	#internal.panel[#PB_Configuration.itLoaderPbID].boSemiAMode := #internal.boManSelOnPressL OR #internal.boSetupSelOnPressL OR #internal.boManSelOnPressR OR #internal.boSetupSelOnPressR;
	#internal.panel[#PB_Configuration.itGTSPbID].boSemiAMode := #internal.boManSelOnPressL OR #internal.boSetupSelOnPressL OR #internal.boManSelOnPressR OR #internal.boSetupSelOnPressR;
	#internal.panel[#PB_Configuration.itPressPbID].boSemiAMode := #internal.boManSelOnPressL OR #internal.boSetupSelOnPressL OR #internal.boManSelOnPressR OR #internal.boSetupSelOnPressR;
	#internal.panel[#PB_Configuration.itSegmentsPbID].boSemiAMode := #internal.boManSelOnPressL OR #internal.boSetupSelOnPressL OR #internal.boManSelOnPressR OR #internal.boSetupSelOnPressR;
	#internal.panel[#PB_Configuration.itSqueezePbID].boSemiAMode := #internal.boManSelOnPressL OR #internal.boSetupSelOnPressL OR #internal.boManSelOnPressR OR #internal.boSetupSelOnPressR;
	#internal.panel[#PB_Configuration.itTopRingPbID].boSemiAMode := #internal.boManSelOnPressL OR #internal.boSetupSelOnPressL OR #internal.boManSelOnPressR OR #internal.boSetupSelOnPressR;
	#internal.panel[#PB_Configuration.itBotRingPbID].boSemiAMode := #internal.boManSelOnPressL OR #internal.boSetupSelOnPressL OR #internal.boManSelOnPressR OR #internal.boSetupSelOnPressR;
	#internal.panel[#PB_Configuration.itBeadRingPbID].boSemiAMode := #internal.boManSelOnPressL OR #internal.boSetupSelOnPressL OR #internal.boManSelOnPressR OR #internal.boSetupSelOnPressR;
	#internal.panel[#PB_Configuration.itUnloaderPbID].boSemiAMode := #internal.boManSelOnPressL OR #internal.boSetupSelOnPressL OR #internal.boManSelOnPressR OR #internal.boSetupSelOnPressR;
	#internal.panel[#PB_Configuration.itUnloaderPCIPbID].boSemiAMode := #internal.boManSelOnPressL OR #internal.boSetupSelOnPressL OR #internal.boManSelOnPressR OR #internal.boSetupSelOnPressR;
	#internal.panel[#PB_Configuration.itExitConvPbId].boSemiAMode := #internal.boManSelOnPressL OR #internal.boSetupSelOnPressL OR #internal.boManSelOnPressR OR #internal.boSetupSelOnPressR;
	#internal.panel[#PB_Configuration.itHPUPbID].boSemiAMode := (#internal.boManSelOnPressL OR #internal.boSetupSelOnPressL) AND (#internal.boManSelOnPressR OR #internal.boSetupSelOnPressR);
	#internal.panel[#PB_Configuration.itLoaderPbID].boAutoMode := NOT #internal.panel[#PB_Configuration.itLoaderPbID].boSemiAMode;
	#internal.panel[#PB_Configuration.itGTSPbID].boAutoMode := NOT #internal.panel[#PB_Configuration.itGTSPbID].boSemiAMode;
	#internal.panel[#PB_Configuration.itPressPbID].boAutoMode := NOT #internal.panel[#PB_Configuration.itPressPbID].boSemiAMode;
	#internal.panel[#PB_Configuration.itSegmentsPbID].boAutoMode := NOT #internal.panel[#PB_Configuration.itSegmentsPbID].boSemiAMode;
	#internal.panel[#PB_Configuration.itSqueezePbID].boAutoMode := NOT #internal.panel[#PB_Configuration.itSqueezePbID].boSemiAMode;
	#internal.panel[#PB_Configuration.itTopRingPbID].boAutoMode := NOT #internal.panel[#PB_Configuration.itTopRingPbID].boSemiAMode;
	#internal.panel[#PB_Configuration.itBotRingPbID].boAutoMode := NOT #internal.panel[#PB_Configuration.itBotRingPbID].boSemiAMode;
	#internal.panel[#PB_Configuration.itBeadRingPbID].boAutoMode := NOT #internal.panel[#PB_Configuration.itBeadRingPbID].boSemiAMode;
	#internal.panel[#PB_Configuration.itUnloaderPbID].boAutoMode := NOT #internal.panel[#PB_Configuration.itUnloaderPbID].boSemiAMode;
	#internal.panel[#PB_Configuration.itUnloaderPCIPbID].boAutoMode := NOT #internal.panel[#PB_Configuration.itUnloaderPCIPbID].boSemiAMode;
	#internal.panel[#PB_Configuration.itExitConvPbId].boAutoMode := NOT #internal.panel[#PB_Configuration.itExitConvPbId].boSemiAMode;
	#internal.panel[#PB_Configuration.itHPUPbID].boAutoMode := NOT #internal.panel[#PB_Configuration.itHPUPbID].boSemiAMode;
	#internal.panel[#PB_Configuration.itShapingPbID].boSemiAMode := #internal.boManSelOnHeatingL OR #internal.boSetupSelOnHeatingL OR #internal.boManSelOnHeatingR OR #internal.boSetupSelOnHeatingR;
	#internal.panel[#PB_Configuration.itDrainPbID].boSemiAMode := #internal.boManSelOnHeatingL OR #internal.boSetupSelOnHeatingL OR #internal.boManSelOnHeatingR OR #internal.boSetupSelOnHeatingR;
	#internal.panel[#PB_Configuration.itVacuumPbID].boSemiAMode := #internal.boManSelOnHeatingL OR #internal.boSetupSelOnHeatingL OR #internal.boManSelOnHeatingR OR #internal.boSetupSelOnHeatingR;
	#internal.panel[#PB_Configuration.itExtHeatingPbID].boSemiAMode := #internal.boManSelOnHeatingL OR #internal.boSetupSelOnHeatingL OR #internal.boManSelOnHeatingR OR #internal.boSetupSelOnHeatingR;
	#internal.panel[#PB_Configuration.itShapingPbID].boAutoMode := NOT #internal.panel[#PB_Configuration.itShapingPbID].boSemiAMode;
	#internal.panel[#PB_Configuration.itDrainPbID].boAutoMode := NOT #internal.panel[#PB_Configuration.itDrainPbID].boSemiAMode;
	#internal.panel[#PB_Configuration.itVacuumPbID].boAutoMode := NOT #internal.panel[#PB_Configuration.itVacuumPbID].boSemiAMode;
	#internal.panel[#PB_Configuration.itExtHeatingPbID].boAutoMode := NOT #internal.panel[#PB_Configuration.itExtHeatingPbID].boSemiAMode;
	END_REGION

	//=======================================================================================================================================
	//            READ INPUTS FROM KP32F
	//=======================================================================================================================================
	REGION READ INPUTS FROM KP32F
	    // Enable test lamp button
	    #internal.panel[#PB_Configuration.itLampTestPbID].boEnable := TRUE;

	    IF NOT "SYS_SimulationActive" THEN
	        // Read push buttons from 0 to 15
	        #readWriteData(itDeviceNumber := #itKP32DeviceNumber,
	                       uiPNIO_SysID := #uiPNIOSysID,
	                       uiSlotNumber := 1,
	                       uiSubSlotNumber := 0,
	                       bo0read_1write := FALSE,
	                       vaModuleSlotData := #internal.buttons0_15);
	        // Read push buttons from 16 to 31
	        #readWriteData(itDeviceNumber := #itKP32DeviceNumber,
	                       uiPNIO_SysID := #uiPNIOSysID,
	                       uiSlotNumber := 2,
	                       uiSubSlotNumber := 0,
	                       bo0read_1write := FALSE,
	                       vaModuleSlotData := #internal.buttons16_31);
	    END_IF;

	    // KP32F management of lamps and buttons
	    FOR #itPushButtonIndexTemp := 0 TO 31 DO

	        (*
	        Push buttons lamp management:
	                OUT:   red      green      blue
	        COLOUR:
	            red         1         0         0
	            green       0         1         0
	            blue        0         0         1
	            yellow      1         1         0
	            white       1         1         1
	            OFF         0         0         0
	            OFF         0         1         1
	            OFF         1         0         1

	        Push buttons order in the panel:
	            07  06  05  04  03  02  01  00
	            15  14  13  12  11  10  09  08
	            23  22  21  20  19  18  17  16
	            31  30  29  28  27  26  25  24
	        *)
	        // Read command button
	        IF NOT "SYS_SimulationActive" THEN
	            CASE #itPushButtonIndexTemp OF
	                0:
	                    #internal.panel[#itPushButtonIndexTemp].boCmdOn := #internal.buttons0_15.PB00;
	                1:
	                    #internal.panel[#itPushButtonIndexTemp].boCmdOn := #internal.buttons0_15.PB01;
	                2:
	                    #internal.panel[#itPushButtonIndexTemp].boCmdOn := #internal.buttons0_15.PB02;
	                3:
	                    #internal.panel[#itPushButtonIndexTemp].boCmdOn := #internal.buttons0_15.PB03;
	                4:
	                    #internal.panel[#itPushButtonIndexTemp].boCmdOn := #internal.buttons0_15.PB04;
	                5:
	                    #internal.panel[#itPushButtonIndexTemp].boCmdOn := #internal.buttons0_15.PB05;
	                6:
	                    #internal.panel[#itPushButtonIndexTemp].boCmdOn := #internal.buttons0_15.PB06;
	                7:
	                    #internal.panel[#itPushButtonIndexTemp].boCmdOn := #internal.buttons0_15.PB07;
	                8:
	                    #internal.panel[#itPushButtonIndexTemp].boCmdOn := #internal.buttons0_15.PB08;
	                9:
	                    #internal.panel[#itPushButtonIndexTemp].boCmdOn := #internal.buttons0_15.PB09;
	                10:
	                    #internal.panel[#itPushButtonIndexTemp].boCmdOn := #internal.buttons0_15.PB10;
	                11:
	                    #internal.panel[#itPushButtonIndexTemp].boCmdOn := #internal.buttons0_15.PB11;
	                12:
	                    #internal.panel[#itPushButtonIndexTemp].boCmdOn := #internal.buttons0_15.PB12;
	                13:
	                    #internal.panel[#itPushButtonIndexTemp].boCmdOn := #internal.buttons0_15.PB13;
	                14:
	                    #internal.panel[#itPushButtonIndexTemp].boCmdOn := #internal.buttons0_15.PB14;
	                15:
	                    #internal.panel[#itPushButtonIndexTemp].boCmdOn := #internal.buttons0_15.PB15;
	                16:
	                    #internal.panel[#itPushButtonIndexTemp].boCmdOn := #internal.buttons16_31.PB16;
	                17:
	                    #internal.panel[#itPushButtonIndexTemp].boCmdOn := #internal.buttons16_31.PB17;
	                18:
	                    #internal.panel[#itPushButtonIndexTemp].boCmdOn := #internal.buttons16_31.PB18;
	                19:
	                    #internal.panel[#itPushButtonIndexTemp].boCmdOn := #internal.buttons16_31.PB19;
	                20:
	                    #internal.panel[#itPushButtonIndexTemp].boCmdOn := #internal.buttons16_31.PB20;
	                21:
	                    #internal.panel[#itPushButtonIndexTemp].boCmdOn := #internal.buttons16_31.PB21;
	                22:
	                    #internal.panel[#itPushButtonIndexTemp].boCmdOn := #internal.buttons16_31.PB22;
	                23:
	                    #internal.panel[#itPushButtonIndexTemp].boCmdOn := #internal.buttons16_31.PB23;
	                24:
	                    #internal.panel[#itPushButtonIndexTemp].boCmdOn := #internal.buttons16_31.PB24;
	                25:
	                    #internal.panel[#itPushButtonIndexTemp].boCmdOn := #internal.buttons16_31.PB25;
	                26:
	                    #internal.panel[#itPushButtonIndexTemp].boCmdOn := #internal.buttons16_31.PB26;
	                27:
	                    #internal.panel[#itPushButtonIndexTemp].boCmdOn := #internal.buttons16_31.PB27;
	                28:
	                    #internal.panel[#itPushButtonIndexTemp].boCmdOn := #internal.buttons16_31.PB28;
	                29:
	                    #internal.panel[#itPushButtonIndexTemp].boCmdOn := #internal.buttons16_31.PB29;
	                30:
	                    #internal.panel[#itPushButtonIndexTemp].boCmdOn := #internal.buttons16_31.PB30;
	                31:
	                    #internal.panel[#itPushButtonIndexTemp].boCmdOn := #internal.buttons16_31.PB31;
	                ELSE
	                    #internal.panel[#itPushButtonIndexTemp].boCmdOn := FALSE;
	            END_CASE;
	        ELSE
	            #internal.panel[#itPushButtonIndexTemp].boCmdOn := #internal.simulation[#itPushButtonIndexTemp].boPB;
	        END_IF;
	        #internal.panel[#itPushButtonIndexTemp].boCmdWrong := FALSE;
	        IF NOT #internal.panel[#itPushButtonIndexTemp].boEnable OR #boChgOfModeFiltTemp THEN
	            IF #internal.panel[#itPushButtonIndexTemp].boCmdOn AND NOT #boChgOfModeFiltTemp THEN
	                #internal.panel[#itPushButtonIndexTemp].boCmdWrong := TRUE;
	                #boWrongPushCmdTemp := TRUE;
	            END_IF;
	            #internal.panel[#itPushButtonIndexTemp].boCmdOn := FALSE;
	            #internal.panel[#itPushButtonIndexTemp].boSelect := FALSE;
	        END_IF;
	        #internal.panel[#itPushButtonIndexTemp].boCmdRE := #internal.panel[#itPushButtonIndexTemp].boCmdOn AND NOT #internal.panel[#itPushButtonIndexTemp].boCmdMem;
	        #internal.panel[#itPushButtonIndexTemp].boCmdFE := NOT #internal.panel[#itPushButtonIndexTemp].boCmdOn AND #internal.panel[#itPushButtonIndexTemp].boCmdMem;
	        #internal.panel[#itPushButtonIndexTemp].boCmdMem := #internal.panel[#itPushButtonIndexTemp].boCmdOn;

	        IF (#internal.panel[#itPushButtonIndexTemp].itPBType = #PB_EQUIPMENT) AND #internal.panel[#itPushButtonIndexTemp].boCmdRE THEN
	            #internal.panel[#itPushButtonIndexTemp].boSelect := NOT #internal.panel[#itPushButtonIndexTemp].boSelect;
	            FOR #itPushButtonIndex2Temp := 0 TO 31 DO
	                IF (#internal.panel[#itPushButtonIndex2Temp].itPBType = #PB_EQUIPMENT) AND (#itPushButtonIndexTemp <> #itPushButtonIndex2Temp) THEN
	                    #internal.panel[#itPushButtonIndex2Temp].boSelect := FALSE;
	                END_IF;
	            END_FOR;
	            #boResetPBsStatesTemp := TRUE;
	        END_IF;

	    END_FOR;
	END_REGION


	//=======================================================================================================================================
	//            CAVITY SELECTION
	//=======================================================================================================================================
	REGION CAVITY SELECTION
	    #internal.panel[#PB_Configuration.itLeftSelPbID].boEnable := TRUE;
	    #internal.panel[#PB_Configuration.itRightSelPbID].boEnable := TRUE;
	    #internal.panel[#PB_Configuration.itLeftSelPbID].boAborted := FALSE;
	    #internal.panel[#PB_Configuration.itRightSelPbID].boAborted := FALSE;
	    #internal.panel[#PB_Configuration.itLeftSelPbID].boHeld := FALSE;
	    #internal.panel[#PB_Configuration.itRightSelPbID].boHeld := FALSE;

	    #internal.panel[#PB_Configuration.itOnOffSelPbID].boOnPos := FALSE;
	    #internal.panel[#PB_Configuration.itInCmdPbID].boOnPos := FALSE;
	    #internal.panel[#PB_Configuration.itOutCmdPbID].boOnPos := FALSE;
	    #internal.panel[#PB_Configuration.itUpCmdPbID].boOnPos := FALSE;
	    #internal.panel[#PB_Configuration.itDownCmdPbID].boOnPos := FALSE;
	    #internal.panel[#PB_Configuration.itRetractCmdPbID].boOnPos := FALSE;
	    #internal.panel[#PB_Configuration.itExpandCmdPbID].boOnPos := FALSE;
	    #internal.panel[#PB_Configuration.itUnlockCmdPbID].boOnPos := FALSE;
	    #internal.panel[#PB_Configuration.itLockCmdPbID].boOnPos := FALSE;

	    //#########################################
	    //#########################################
	    IF #boManSelCavityL THEN
	        #itLeftSelectorStateTemp := 1;
	    ELSIF #boAutoSelpCavityL THEN
	        #itLeftSelectorStateTemp := 2;
	    ELSE
	        #itLeftSelectorStateTemp := 0;
	    END_IF;

	    IF #boManSelCavityR THEN
	        #itRightSelectorStateTemp := 1;
	    ELSIF #boAutoSelpCavityR THEN
	        #itRightSelectorStateTemp := 2;
	    ELSE
	        #itRightSelectorStateTemp := 0;
	    END_IF;

	    #boLeftSelUpdateTemp := #itLeftSelectorStateTemp <> #internal.itLeftSelectorState;
	    #boRightSelUpdateTemp := #itRightSelectorStateTemp <> #internal.itRightSelectorState;
	    IF NOT #internal.chgModeTOF.Q THEN
	        #internal.itLeftSelectorState := #itLeftSelectorStateTemp;
	        #internal.itRightSelectorState := #itRightSelectorStateTemp;
	    END_IF;
	    //#########################################
	    //#########################################
	    IF NOT #internal.panel[#PB_Configuration.itLeftSelPbID].boSelect AND NOT #internal.panel[#PB_Configuration.itRightSelPbID].boSelect THEN
	        #internal.panel[#PB_Configuration.itLeftSelPbID].boSelect := TRUE;
	        #internal.panel[#PB_Configuration.itRightSelPbID].boSelect := TRUE;
	    ELSIF (#internal.panel[#PB_Configuration.itLeftSelPbID].boCmdRE OR #boLeftSelUpdateTemp) THEN //AND NOT (unitL."to".boGymActivated) THEN // OR _internal.panel[itGymPbID].boSelect) THEN
	        IF #internal.panel[#PB_Configuration.itLeftSelPbID].boSelect THEN
	            #internal.panel[#PB_Configuration.itRightSelPbID].boSelect := FALSE;
	        ELSE
	            #internal.panel[#PB_Configuration.itLeftSelPbID].boSelect := TRUE;
	        END_IF;
	    ELSIF (#internal.panel[#PB_Configuration.itRightSelPbID].boCmdRE OR #boRightSelUpdateTemp) THEN //AND NOT (unitR."to".boGymActivated) THEN // OR _internal.panel[itGymPbID].boSelect) THEN
	        IF #internal.panel[#PB_Configuration.itRightSelPbID].boSelect THEN
	            #internal.panel[#PB_Configuration.itLeftSelPbID].boSelect := FALSE;
	        ELSE
	            #internal.panel[#PB_Configuration.itRightSelPbID].boSelect := TRUE;
	        END_IF;
	    END_IF;
	    IF #internal.panel[#PB_Configuration.itShapingPbID].boSelect OR #internal.panel[#PB_Configuration.itDrainPbID].boSelect OR #internal.panel[#PB_Configuration.itVacuumPbID].boSelect THEN
	        IF #unitL."to".boMoldDisabled AND (#internal.boManSelOnHeatingL OR #internal.boSetupProcActiveL) THEN
	            #internal.panel[#PB_Configuration.itLeftSelPbID].boSelect := FALSE;
	        END_IF;
	        IF #unitR."to".boMoldDisabled AND (#internal.boManSelOnHeatingR OR #internal.boSetupProcActiveR) THEN
	            #internal.panel[#PB_Configuration.itRightSelPbID].boSelect := FALSE;
	        END_IF;
	    END_IF;
	END_REGION

	REGION EQ
	    #internal.panel[#PB_Configuration.itUnitPbID].boEnable := FALSE;
	    #internal.panel[#PB_Configuration.itPickupPbID].boEnable := FALSE;

	    #internal.panel[#PB_Configuration.itUnitPbID].boAborted := FALSE;
	    #internal.panel[#PB_Configuration.itPickupPbID].boAborted := FALSE;
	    #internal.panel[#PB_Configuration.itUnitPbID].boHeld := FALSE;

	    #internal.panel[#PB_Configuration.itGTSPbID].boAborted := FALSE;
	    #internal.panel[#PB_Configuration.itGTSPbID].boHeld := FALSE;

	    #internal.panel[#PB_Configuration.itLoaderPbID].boAborted := FALSE;
	    #internal.panel[#PB_Configuration.itLoaderPbID].boHeld := FALSE;

	    #internal.panel[#PB_Configuration.itPressPbID].boAborted := FALSE;
	    #internal.panel[#PB_Configuration.itPressPbID].boHeld := FALSE;

	    #internal.panel[#PB_Configuration.itTopRingPbID].boAborted := FALSE;
	    #internal.panel[#PB_Configuration.itTopRingPbID].boHeld := FALSE;
	    #internal.panel[#PB_Configuration.itBotRingPbID].boAborted := FALSE;
	    #internal.panel[#PB_Configuration.itBotRingPbID].boHeld := FALSE;
	    #internal.panel[#PB_Configuration.itBeadRingPbID].boAborted := FALSE;
	    #internal.panel[#PB_Configuration.itBeadRingPbID].boHeld := FALSE;

	    #internal.panel[#PB_Configuration.itUnloaderPbID].boAborted := FALSE;
	    #internal.panel[#PB_Configuration.itUnloaderPbID].boHeld := FALSE;
	    #internal.panel[#PB_Configuration.itUnloaderPCIPbID].boAborted := FALSE;
	    #internal.panel[#PB_Configuration.itUnloaderPCIPbID].boHeld := FALSE;

	    #internal.panel[#PB_Configuration.itExitConvPbId].boAborted := FALSE;
	    #internal.panel[#PB_Configuration.itExitConvPbId].boHeld := FALSE;
	END_REGION

	//=======================================================================================================================================
	//            PRODUCTION PROGRAM SEMI-AUTO
	//=======================================================================================================================================
	REGION PRODUCTION PROGRAM SEMI-AUTO
	    REGION LOADERS & MGTS
	        IF (#internal.boManSelOnPressL OR #internal.boSetupSelOnPressL OR #internal.boSetupProcActiveL) AND #internal.panel[#PB_Configuration.itLeftSelPbID].boSelect THEN
	            // Enable push-buttons
	            #internal.panel[#PB_Configuration.itLoaderPbID].boEnable := TRUE;

	            // Modules fault & warning
	            #internal.panel[#PB_Configuration.itLoaderPbID].boAborted := #EQloaderL."to".boStatusAbortedEQ OR #EQloaderL."to".boStatusAbortedSwing OR #EQloaderL."to".boStatusAbortedUDMove OR #EQloaderL."to".boStatusAbortedPaddles;
	            #internal.panel[#PB_Configuration.itLoaderPbID].boHeld := #EQloaderL."to".boStatusHeldEQ OR #EQloaderL."to".boStatusHeldSwing OR #EQloaderL."to".boStatusHeldUDMove OR #EQloaderL."to".boStatusHeldPaddles;

	            // Loaders: manual commands
	            IF #internal.panel[#PB_Configuration.itLoaderPbID].boSelect THEN
	                #internal.panel[#PB_Configuration.itLeftSelPbID].boAborted := #EQloaderL."to".boStatusAbortedEQ OR #EQloaderL."to".boStatusAbortedSwing OR #EQloaderL."to".boStatusAbortedUDMove OR #EQloaderL."to".boStatusAbortedPaddles;
	                #internal.panel[#PB_Configuration.itLeftSelPbID].boHeld := #EQloaderL."to".boStatusHeldEQ OR #EQloaderL."to".boStatusHeldSwing OR #EQloaderL."to".boStatusHeldUDMove OR #EQloaderL."to".boStatusHeldPaddles;

	                #internal.panel[#PB_Configuration.itInCmdPbID].boOnPos := #EQloaderL."to".boPosSwingIn;
	                #internal.panel[#PB_Configuration.itOutCmdPbID].boOnPos := #EQloaderL."to".boPosSwingOut;
	                #internal.panel[#PB_Configuration.itUpCmdPbID].boOnPos := #EQloaderL."to".boPosLoaderUp;
	                #internal.panel[#PB_Configuration.itDownCmdPbID].boOnPos := #EQloaderL."to".boPosLoaderDown;
	                #internal.panel[#PB_Configuration.itRetractCmdPbID].boOnPos := #EQloaderL."to".boPosPaddlesRet;
	                #internal.panel[#PB_Configuration.itExpandCmdPbID].boOnPos := #EQloaderL."to".boPosPaddlesExp;

	                #internal.panel[#PB_Configuration.itInCmdPbID].boMoving := #EQloaderL."to".boMoveSwingIn;
	                #internal.panel[#PB_Configuration.itOutCmdPbID].boMoving := #EQloaderL."to".boMoveSwingOut;
	                #internal.panel[#PB_Configuration.itUpCmdPbID].boMoving := #EQloaderL."to".boMoveLoaderUp;
	                #internal.panel[#PB_Configuration.itDownCmdPbID].boMoving := #EQloaderL."to".boMoveLoaderDown;
	                #internal.panel[#PB_Configuration.itRetractCmdPbID].boMoving := #EQloaderL."to".boMovePaddlesRet;
	                #internal.panel[#PB_Configuration.itExpandCmdPbID].boMoving := #EQloaderL."to".boMovePaddlesExp;

	                #internal.panel[#PB_Configuration.itInCmdPbID].boEnable := #EQloaderL."to".boEnaSwingIn OR #internal.panel[#PB_Configuration.itInCmdPbID].boOnPos OR #internal.panel[#PB_Configuration.itInCmdPbID].boMoving;
	                #internal.panel[#PB_Configuration.itOutCmdPbID].boEnable := #EQloaderL."to".boEnaSwingOut OR #internal.panel[#PB_Configuration.itOutCmdPbID].boOnPos OR #internal.panel[#PB_Configuration.itOutCmdPbID].boMoving;
	                #internal.panel[#PB_Configuration.itUpCmdPbID].boEnable := #EQloaderL."to".boEnaLoaderUp OR #internal.panel[#PB_Configuration.itUpCmdPbID].boOnPos OR #internal.panel[#PB_Configuration.itUpCmdPbID].boMoving;
	                #internal.panel[#PB_Configuration.itDownCmdPbID].boEnable := #EQloaderL."to".boEnaLoaderDown OR #internal.panel[#PB_Configuration.itDownCmdPbID].boOnPos OR #internal.panel[#PB_Configuration.itDownCmdPbID].boMoving;
	                #internal.panel[#PB_Configuration.itRetractCmdPbID].boEnable := #EQloaderL."to".boEnaPaddlesRet OR #internal.panel[#PB_Configuration.itRetractCmdPbID].boOnPos OR #internal.panel[#PB_Configuration.itRetractCmdPbID].boMoving;
	                #internal.panel[#PB_Configuration.itExpandCmdPbID].boEnable := #EQloaderL."to".boEnaPaddlesExp OR #internal.panel[#PB_Configuration.itExpandCmdPbID].boOnPos OR #internal.panel[#PB_Configuration.itExpandCmdPbID].boMoving;

	                #EQloaderL.from.boCmdSwingIn := #internal.panel[#PB_Configuration.itInCmdPbID].boCmdOn;
	                #EQloaderL.from.boCmdSwingOut := #internal.panel[#PB_Configuration.itOutCmdPbID].boCmdOn;
	                #EQloaderL.from.boCmdUDMoveDown := #internal.panel[#PB_Configuration.itDownCmdPbID].boCmdOn;
	                #EQloaderL.from.boCmdUDMoveUp := #internal.panel[#PB_Configuration.itUpCmdPbID].boCmdOn;
	                #EQloaderL.from.boCmdPaddlesExp := #internal.panel[#PB_Configuration.itExpandCmdPbID].boCmdOn;
	                #EQloaderL.from.boCmdPaddlesRet := #internal.panel[#PB_Configuration.itRetractCmdPbID].boCmdOn;
	            END_IF;

	            // Enable push-buttons
	            #internal.panel[#PB_Configuration.itGTSPbID].boEnable := TRUE;

	            // Modules fault & warning
	            #internal.panel[#PB_Configuration.itGTSPbID].boAborted := #EQgtsL."to".boStatusAbortedEQ OR #EQgtsL."to".boStatusAbortedSwing;
	            #internal.panel[#PB_Configuration.itGTSPbID].boHeld := #EQgtsL."to".boStatusHeldEQ OR #EQgtsL."to".boStatusHeldSwing;

	            // GTS: manual commands
	            IF #internal.panel[#PB_Configuration.itGTSPbID].boSelect THEN
	                #internal.panel[#PB_Configuration.itLeftSelPbID].boAborted := #EQgtsL."to".boStatusAbortedEQ OR #EQgtsL."to".boStatusAbortedSwing;
	                #internal.panel[#PB_Configuration.itLeftSelPbID].boHeld := #EQgtsL."to".boStatusHeldEQ OR #EQgtsL."to".boStatusHeldSwing;

	                #internal.panel[#PB_Configuration.itInCmdPbID].boOnPos := #EQgtsL."to".boPosSwingIn;
	                #internal.panel[#PB_Configuration.itOutCmdPbID].boOnPos := #EQgtsL."to".boPosSwingOut;

	                #internal.panel[#PB_Configuration.itInCmdPbID].boMoving := #EQgtsL."to".boMoveSwingIn;
	                #internal.panel[#PB_Configuration.itOutCmdPbID].boMoving := #EQgtsL."to".boMoveSwingOut;

	                #internal.panel[#PB_Configuration.itInCmdPbID].boEnable := #EQgtsL."to".boEnaSwingIn OR #internal.panel[#PB_Configuration.itInCmdPbID].boOnPos OR #internal.panel[#PB_Configuration.itInCmdPbID].boMoving;
	                #internal.panel[#PB_Configuration.itOutCmdPbID].boEnable := #EQgtsL."to".boEnaSwingOut OR #internal.panel[#PB_Configuration.itOutCmdPbID].boOnPos OR #internal.panel[#PB_Configuration.itOutCmdPbID].boMoving;

	                #EQgtsL.from.boCmdSwingIn := #internal.panel[#PB_Configuration.itInCmdPbID].boCmdOn;
	                #EQgtsL.from.boCmdSwingOut := #internal.panel[#PB_Configuration.itOutCmdPbID].boCmdOn;
	            END_IF;
	        END_IF;

	        IF (#internal.boManSelOnPressR OR #internal.boSetupSelOnPressR OR #internal.boSetupProcActiveR) AND #internal.panel[#PB_Configuration.itRightSelPbID].boSelect THEN
	            // Enable push-buttons
	            #internal.panel[#PB_Configuration.itLoaderPbID].boEnable := TRUE;

	            // Modules fault & warning
	            #internal.panel[#PB_Configuration.itLoaderPbID].boAborted := #EQloaderR."to".boStatusAbortedEQ OR #EQloaderR."to".boStatusAbortedSwing OR #EQloaderR."to".boStatusAbortedUDMove OR #EQloaderR."to".boStatusAbortedPaddles;
	            #internal.panel[#PB_Configuration.itLoaderPbID].boHeld := #EQloaderR."to".boStatusHeldEQ OR #EQloaderR."to".boStatusHeldSwing OR #EQloaderR."to".boStatusHeldUDMove OR #EQloaderR."to".boStatusHeldPaddles;

	            // Loaders: manual commands
	            IF #internal.panel[#PB_Configuration.itLoaderPbID].boSelect THEN

	                #internal.panel[#PB_Configuration.itRightSelPbID].boAborted := #EQloaderR."to".boStatusAbortedEQ OR #EQloaderR."to".boStatusAbortedSwing OR #EQloaderR."to".boStatusAbortedUDMove OR #EQloaderR."to".boStatusAbortedPaddles;
	                #internal.panel[#PB_Configuration.itRightSelPbID].boHeld := #EQloaderR."to".boStatusHeldEQ OR #EQloaderR."to".boStatusHeldSwing OR #EQloaderR."to".boStatusHeldUDMove OR #EQloaderR."to".boStatusHeldPaddles;

	                #internal.panel[#PB_Configuration.itInCmdPbID].boOnPos := #EQloaderR."to".boPosSwingIn;
	                #internal.panel[#PB_Configuration.itOutCmdPbID].boOnPos := #EQloaderR."to".boPosSwingOut;
	                #internal.panel[#PB_Configuration.itUpCmdPbID].boOnPos := #EQloaderR."to".boPosLoaderUp;
	                #internal.panel[#PB_Configuration.itDownCmdPbID].boOnPos := #EQloaderR."to".boPosLoaderDown;
	                #internal.panel[#PB_Configuration.itRetractCmdPbID].boOnPos := #EQloaderR."to".boPosPaddlesRet;
	                #internal.panel[#PB_Configuration.itExpandCmdPbID].boOnPos := #EQloaderR."to".boPosPaddlesExp;

	                #internal.panel[#PB_Configuration.itInCmdPbID].boMoving := #EQloaderR."to".boMoveSwingIn;
	                #internal.panel[#PB_Configuration.itOutCmdPbID].boMoving := #EQloaderR."to".boMoveSwingOut;
	                #internal.panel[#PB_Configuration.itUpCmdPbID].boMoving := #EQloaderR."to".boMoveLoaderUp;
	                #internal.panel[#PB_Configuration.itDownCmdPbID].boMoving := #EQloaderR."to".boMoveLoaderDown;
	                #internal.panel[#PB_Configuration.itRetractCmdPbID].boMoving := #EQloaderR."to".boMovePaddlesRet;
	                #internal.panel[#PB_Configuration.itExpandCmdPbID].boMoving := #EQloaderR."to".boMovePaddlesExp;

	                #internal.panel[#PB_Configuration.itInCmdPbID].boEnable := #EQloaderR."to".boEnaSwingIn OR #internal.panel[#PB_Configuration.itInCmdPbID].boOnPos OR #internal.panel[#PB_Configuration.itInCmdPbID].boMoving;
	                #internal.panel[#PB_Configuration.itOutCmdPbID].boEnable := #EQloaderR."to".boEnaSwingOut OR #internal.panel[#PB_Configuration.itOutCmdPbID].boOnPos OR #internal.panel[#PB_Configuration.itOutCmdPbID].boMoving;
	                #internal.panel[#PB_Configuration.itUpCmdPbID].boEnable := #EQloaderR."to".boEnaLoaderUp OR #internal.panel[#PB_Configuration.itUpCmdPbID].boOnPos OR #internal.panel[#PB_Configuration.itUpCmdPbID].boMoving;
	                #internal.panel[#PB_Configuration.itDownCmdPbID].boEnable := #EQloaderR."to".boEnaLoaderDown OR #internal.panel[#PB_Configuration.itDownCmdPbID].boOnPos OR #internal.panel[#PB_Configuration.itDownCmdPbID].boMoving;
	                #internal.panel[#PB_Configuration.itRetractCmdPbID].boEnable := #EQloaderR."to".boEnaPaddlesRet OR #internal.panel[#PB_Configuration.itRetractCmdPbID].boOnPos OR #internal.panel[#PB_Configuration.itRetractCmdPbID].boMoving;
	                #internal.panel[#PB_Configuration.itExpandCmdPbID].boEnable := #EQloaderR."to".boEnaPaddlesExp OR #internal.panel[#PB_Configuration.itExpandCmdPbID].boOnPos OR #internal.panel[#PB_Configuration.itExpandCmdPbID].boMoving;

	                #EQloaderR.from.boCmdSwingIn := #internal.panel[#PB_Configuration.itInCmdPbID].boCmdOn;
	                #EQloaderR.from.boCmdSwingOut := #internal.panel[#PB_Configuration.itOutCmdPbID].boCmdOn;
	                #EQloaderR.from.boCmdUDMoveDown := #internal.panel[#PB_Configuration.itDownCmdPbID].boCmdOn;
	                #EQloaderR.from.boCmdUDMoveUp := #internal.panel[#PB_Configuration.itUpCmdPbID].boCmdOn;
	                #EQloaderR.from.boCmdPaddlesExp := #internal.panel[#PB_Configuration.itExpandCmdPbID].boCmdOn;
	                #EQloaderR.from.boCmdPaddlesRet := #internal.panel[#PB_Configuration.itRetractCmdPbID].boCmdOn;
	            END_IF;

	            // Enable push-buttons
	            #internal.panel[#PB_Configuration.itGTSPbID].boEnable := TRUE;

	            // Modules fault & warning
	            #internal.panel[#PB_Configuration.itGTSPbID].boAborted := #EQgtsR."to".boStatusAbortedEQ OR #EQgtsR."to".boStatusAbortedSwing;
	            #internal.panel[#PB_Configuration.itGTSPbID].boHeld := #EQgtsR."to".boStatusHeldEQ OR #EQgtsR."to".boStatusHeldSwing;

	            // GTS: manual commands
	            IF #internal.panel[#PB_Configuration.itGTSPbID].boSelect THEN
	                #internal.panel[#PB_Configuration.itRightSelPbID].boAborted := #EQgtsR."to".boStatusAbortedEQ OR #EQgtsR."to".boStatusAbortedSwing;
	                #internal.panel[#PB_Configuration.itRightSelPbID].boHeld := #EQgtsR."to".boStatusHeldEQ OR #EQgtsR."to".boStatusHeldSwing;

	                #internal.panel[#PB_Configuration.itInCmdPbID].boOnPos := #EQgtsR."to".boPosSwingIn;
	                #internal.panel[#PB_Configuration.itOutCmdPbID].boOnPos := #EQgtsR."to".boPosSwingOut;

	                #internal.panel[#PB_Configuration.itInCmdPbID].boMoving := #EQgtsR."to".boMoveSwingIn;
	                #internal.panel[#PB_Configuration.itOutCmdPbID].boMoving := #EQgtsR."to".boMoveSwingOut;

	                #internal.panel[#PB_Configuration.itInCmdPbID].boEnable := #EQgtsR."to".boEnaSwingIn OR #internal.panel[#PB_Configuration.itInCmdPbID].boOnPos OR #internal.panel[#PB_Configuration.itInCmdPbID].boMoving;
	                #internal.panel[#PB_Configuration.itOutCmdPbID].boEnable := #EQgtsR."to".boEnaSwingOut OR #internal.panel[#PB_Configuration.itOutCmdPbID].boOnPos OR #internal.panel[#PB_Configuration.itOutCmdPbID].boMoving;

	                #EQgtsR.from.boCmdSwingIn := #internal.panel[#PB_Configuration.itInCmdPbID].boCmdOn;
	                #EQgtsR.from.boCmdSwingOut := #internal.panel[#PB_Configuration.itOutCmdPbID].boCmdOn;
	            END_IF;
	        END_IF;

	        IF ((#internal.boManSelOnPressL OR #internal.boSetupSelOnPressL OR #internal.boSetupProcActiveL) AND #internal.panel[#PB_Configuration.itLeftSelPbID].boSelect) AND
	            ((#internal.boManSelOnPressR OR #internal.boSetupSelOnPressR OR #internal.boSetupProcActiveR) AND #internal.panel[#PB_Configuration.itRightSelPbID].boSelect) THEN
	            // Enable push-buttons
	            #internal.panel[#PB_Configuration.itLoaderPbID].boEnable := TRUE;

	            // Modules fault & warning
	            #internal.panel[#PB_Configuration.itLoaderPbID].boAborted := #EQloaderL."to".boStatusAbortedEQ OR #EQloaderL."to".boStatusAbortedSwing OR #EQloaderL."to".boStatusAbortedUDMove OR #EQloaderL."to".boStatusAbortedPaddles OR
	            #EQloaderR."to".boStatusAbortedEQ OR #EQloaderR."to".boStatusAbortedSwing OR #EQloaderR."to".boStatusAbortedUDMove OR #EQloaderR."to".boStatusAbortedPaddles;
	            #internal.panel[#PB_Configuration.itLoaderPbID].boHeld := #EQloaderR."to".boStatusHeldEQ OR #EQloaderR."to".boStatusHeldSwing OR #EQloaderR."to".boStatusHeldUDMove OR #EQloaderR."to".boStatusHeldPaddles OR
	            #EQloaderR."to".boStatusHeldEQ OR #EQloaderR."to".boStatusHeldSwing OR #EQloaderR."to".boStatusHeldUDMove OR #EQloaderR."to".boStatusHeldPaddles;

	            // Loaders: manual commands
	            IF #internal.panel[#PB_Configuration.itLoaderPbID].boSelect THEN
	                #internal.panel[#PB_Configuration.itInCmdPbID].boOnPos := #EQloaderL."to".boPosSwingIn AND #EQloaderR."to".boPosSwingIn;
	                #internal.panel[#PB_Configuration.itOutCmdPbID].boOnPos := #EQloaderL."to".boPosSwingOut AND #EQloaderR."to".boPosSwingOut;
	                #internal.panel[#PB_Configuration.itUpCmdPbID].boOnPos := #EQloaderL."to".boPosLoaderUp AND #EQloaderR."to".boPosLoaderUp;
	                #internal.panel[#PB_Configuration.itDownCmdPbID].boOnPos := #EQloaderL."to".boPosLoaderDown AND #EQloaderR."to".boPosLoaderDown;
	                #internal.panel[#PB_Configuration.itRetractCmdPbID].boOnPos := #EQloaderL."to".boPosPaddlesRet AND #EQloaderR."to".boPosPaddlesRet;
	                #internal.panel[#PB_Configuration.itExpandCmdPbID].boOnPos := #EQloaderL."to".boPosPaddlesExp AND #EQloaderR."to".boPosPaddlesExp;

	                #internal.panel[#PB_Configuration.itInCmdPbID].boMoving := #EQloaderL."to".boMoveSwingIn OR #EQloaderR."to".boMoveSwingIn;
	                #internal.panel[#PB_Configuration.itOutCmdPbID].boMoving := #EQloaderL."to".boMoveSwingOut OR #EQloaderR."to".boMoveSwingOut;
	                #internal.panel[#PB_Configuration.itUpCmdPbID].boMoving := #EQloaderL."to".boMoveLoaderUp OR #EQloaderR."to".boMoveLoaderUp;
	                #internal.panel[#PB_Configuration.itDownCmdPbID].boMoving := #EQloaderL."to".boMoveLoaderDown OR #EQloaderR."to".boMoveLoaderDown;
	                #internal.panel[#PB_Configuration.itRetractCmdPbID].boMoving := #EQloaderL."to".boMovePaddlesRet OR #EQloaderR."to".boMovePaddlesRet;
	                #internal.panel[#PB_Configuration.itExpandCmdPbID].boMoving := #EQloaderL."to".boMovePaddlesExp OR #EQloaderR."to".boMovePaddlesExp;

	                #internal.panel[#PB_Configuration.itInCmdPbID].boEnable := #EQloaderL."to".boEnaSwingIn OR #EQloaderR."to".boEnaSwingIn OR #internal.panel[#PB_Configuration.itInCmdPbID].boOnPos OR #internal.panel[#PB_Configuration.itInCmdPbID].boMoving;
	                #internal.panel[#PB_Configuration.itOutCmdPbID].boEnable := #EQloaderL."to".boEnaSwingOut OR #EQloaderR."to".boEnaSwingOut OR #internal.panel[#PB_Configuration.itOutCmdPbID].boOnPos OR #internal.panel[#PB_Configuration.itOutCmdPbID].boMoving;
	                #internal.panel[#PB_Configuration.itUpCmdPbID].boEnable := #EQloaderL."to".boEnaLoaderUp OR #EQloaderR."to".boEnaLoaderUp OR #internal.panel[#PB_Configuration.itUpCmdPbID].boOnPos OR #internal.panel[#PB_Configuration.itUpCmdPbID].boMoving;
	                #internal.panel[#PB_Configuration.itDownCmdPbID].boEnable := #EQloaderL."to".boEnaLoaderDown OR #EQloaderR."to".boEnaLoaderDown OR #internal.panel[#PB_Configuration.itDownCmdPbID].boOnPos OR #internal.panel[#PB_Configuration.itDownCmdPbID].boMoving;
	                #internal.panel[#PB_Configuration.itRetractCmdPbID].boEnable := #EQloaderL."to".boEnaPaddlesRet OR #EQloaderR."to".boEnaPaddlesRet OR #internal.panel[#PB_Configuration.itRetractCmdPbID].boOnPos OR #internal.panel[#PB_Configuration.itRetractCmdPbID].boMoving;
	                #internal.panel[#PB_Configuration.itExpandCmdPbID].boEnable := #EQloaderL."to".boEnaPaddlesExp OR #EQloaderR."to".boEnaPaddlesExp OR #internal.panel[#PB_Configuration.itExpandCmdPbID].boOnPos OR #internal.panel[#PB_Configuration.itExpandCmdPbID].boMoving;
	            END_IF;

	            // Enable push-buttons
	            #internal.panel[#PB_Configuration.itGTSPbID].boEnable := TRUE;

	            // Modules fault & warning
	            #internal.panel[#PB_Configuration.itGTSPbID].boAborted := #EQgtsL."to".boStatusAbortedEQ OR #EQgtsL."to".boStatusAbortedSwing OR #EQgtsR."to".boStatusAbortedEQ OR #EQgtsR."to".boStatusAbortedSwing;
	            #internal.panel[#PB_Configuration.itGTSPbID].boHeld := #EQgtsL."to".boStatusHeldEQ OR #EQgtsL."to".boStatusHeldSwing OR #EQgtsR."to".boStatusHeldEQ OR #EQgtsR."to".boStatusHeldSwing;

	            // GTS: manual commands
	            IF #internal.panel[#PB_Configuration.itGTSPbID].boSelect THEN
	                #internal.panel[#PB_Configuration.itInCmdPbID].boOnPos := #EQgtsL."to".boPosSwingIn OR #EQgtsR."to".boPosSwingIn;
	                #internal.panel[#PB_Configuration.itOutCmdPbID].boOnPos := #EQgtsL."to".boPosSwingOut OR #EQgtsR."to".boPosSwingOut;

	                #internal.panel[#PB_Configuration.itInCmdPbID].boMoving := #EQgtsL."to".boMoveSwingIn OR #EQgtsR."to".boMoveSwingIn;
	                #internal.panel[#PB_Configuration.itOutCmdPbID].boMoving := #EQgtsL."to".boMoveSwingOut OR #EQgtsR."to".boMoveSwingOut;

	                #internal.panel[#PB_Configuration.itInCmdPbID].boEnable := #EQgtsL."to".boEnaSwingIn OR #EQgtsR."to".boEnaSwingIn OR #internal.panel[#PB_Configuration.itInCmdPbID].boOnPos OR #internal.panel[#PB_Configuration.itInCmdPbID].boMoving;
	                #internal.panel[#PB_Configuration.itOutCmdPbID].boEnable := #EQgtsL."to".boEnaSwingOut OR #EQgtsR."to".boEnaSwingOut OR #internal.panel[#PB_Configuration.itOutCmdPbID].boOnPos OR #internal.panel[#PB_Configuration.itOutCmdPbID].boMoving;
	            END_IF;
	        END_IF;
	    END_REGION

	    REGION PRESSES
	        IF (#internal.boManSelOnPressL OR #internal.boSetupSelOnPressL OR #internal.boSetupProcActiveL) AND #internal.panel[#PB_Configuration.itLeftSelPbID].boSelect THEN
	            // Enable push-buttons
	            #internal.panel[#PB_Configuration.itPressPbID].boEnable := TRUE;
	            #internal.panel[#PB_Configuration.itSegmentsPbID].boEnable := TRUE;
	            #internal.panel[#PB_Configuration.itSqueezePbID].boEnable := TRUE;

	            // Modules fault & warning
	            #internal.panel[#PB_Configuration.itPressPbID].boAborted := #EQpressL."to".boStatusAbortedEQ OR #EQpressL."to".boStatusAbortedUDMove;
	            #internal.panel[#PB_Configuration.itSegmentsPbID].boAborted := #EQpressL."to".boStatusAbortedSegments;
	            #internal.panel[#PB_Configuration.itSqueezePbID].boAborted := #EQpressL."to".boStatusAbortedSqueeze;
	            #internal.panel[#PB_Configuration.itPressPbID].boHeld := #EQpressL."to".boStatusHeldEQ OR #EQpressL."to".boStatusHeldUDMove;
	            #internal.panel[#PB_Configuration.itSegmentsPbID].boHeld := #EQpressL."to".boStatusHeldSegments;
	            #internal.panel[#PB_Configuration.itSqueezePbID].boHeld := #EQpressL."to".boStatusHeldSqueeze;

	            // Press: manual commands
	            IF #internal.panel[#PB_Configuration.itPressPbID].boSelect THEN
	                #internal.panel[#PB_Configuration.itLeftSelPbID].boAborted := #EQpressL."to".boStatusAbortedEQ OR #EQpressL."to".boStatusAbortedUDMove;
	                #internal.panel[#PB_Configuration.itLeftSelPbID].boHeld := #EQpressL."to".boStatusHeldEQ OR #EQpressL."to".boStatusHeldUDMove;

	                #internal.panel[#PB_Configuration.itUpCmdPbID].boOnPos := #EQpressL."to".boPosUDMoveUp;
	                #internal.panel[#PB_Configuration.itDownCmdPbID].boOnPos := #EQpressL."to".boPosUDMoveDown;
	                #internal.panel[#PB_Configuration.itLockCmdPbID].boOnPos := #EQpressL."to".boPosUDLock;
	                #internal.panel[#PB_Configuration.itUnlockCmdPbID].boOnPos := #EQpressL."to".boPosUDUnlock;
	                #internal.panel[#PB_Configuration.itInCmdPbID].boOnPos := #EQpressL."to".boPosSafetyBarUp;
	                #internal.panel[#PB_Configuration.itOutCmdPbID].boOnPos := #EQpressL."to".boPosSafetyBarDw;

	                #internal.panel[#PB_Configuration.itUpCmdPbID].boMoving := #EQpressL."to".boMoveUDMoveUp;
	                #internal.panel[#PB_Configuration.itDownCmdPbID].boMoving := #EQpressL."to".boMoveUDMoveDown;
	                #internal.panel[#PB_Configuration.itLockCmdPbID].boMoving := #EQpressL."to".boMoveUDLock;
	                #internal.panel[#PB_Configuration.itUnlockCmdPbID].boMoving := #EQpressL."to".boMoveUDUnlock;
	                #internal.panel[#PB_Configuration.itInCmdPbID].boMoving := #EQpressL."to".boMoveSafetyBarUp;
	                #internal.panel[#PB_Configuration.itOutCmdPbID].boMoving := #EQpressL."to".boMoveSafetyBarDw;

	                #internal.panel[#PB_Configuration.itUpCmdPbID].boEnable := #EQpressL."to".boEnaUDMoveUp OR #internal.panel[#PB_Configuration.itUpCmdPbID].boOnPos OR #internal.panel[#PB_Configuration.itUpCmdPbID].boMoving;
	                #internal.panel[#PB_Configuration.itDownCmdPbID].boEnable := #EQpressL."to".boEnaUDMoveDown OR #internal.panel[#PB_Configuration.itDownCmdPbID].boOnPos OR #internal.panel[#PB_Configuration.itDownCmdPbID].boMoving;
	                #internal.panel[#PB_Configuration.itLockCmdPbID].boEnable := #EQpressL."to".boEnaUDLock OR #internal.panel[#PB_Configuration.itLockCmdPbID].boOnPos OR #internal.panel[#PB_Configuration.itLockCmdPbID].boMoving;
	                #internal.panel[#PB_Configuration.itUnlockCmdPbID].boEnable := #EQpressL."to".boEnaUDUnlock OR #internal.panel[#PB_Configuration.itUnlockCmdPbID].boOnPos OR #internal.panel[#PB_Configuration.itUnlockCmdPbID].boMoving;
	                #internal.panel[#PB_Configuration.itInCmdPbID].boEnable := #EQpressL."to".boEnaSafetyBarUp OR #internal.panel[#PB_Configuration.itInCmdPbID].boOnPos OR #internal.panel[#PB_Configuration.itInCmdPbID].boMoving;
	                #internal.panel[#PB_Configuration.itOutCmdPbID].boEnable := #EQpressL."to".boEnaSafetyBarDw OR #internal.panel[#PB_Configuration.itOutCmdPbID].boOnPos OR #internal.panel[#PB_Configuration.itOutCmdPbID].boMoving;

	                #EQpressL.from.boCmdUDMoveDown := #internal.panel[#PB_Configuration.itDownCmdPbID].boCmdOn;
	                #EQpressL.from.boCmdUDMoveUp := #internal.panel[#PB_Configuration.itUpCmdPbID].boCmdOn;
	                #EQpressL.from.boCmdUDLock := #internal.panel[#PB_Configuration.itLockCmdPbID].boCmdOn;
	                #EQpressL.from.boCmdUDUnlock := #internal.panel[#PB_Configuration.itUnlockCmdPbID].boCmdOn;
	                #EQpressL.from.boCmdSafetyBarUp := #internal.panel[#PB_Configuration.itInCmdPbID].boCmdOn;
	                #EQpressL.from.boCmdSafetyBarDown := #internal.panel[#PB_Configuration.itOutCmdPbID].boCmdOn;
	            END_IF;

	            // Segments: manual commands
	            IF #internal.panel[#PB_Configuration.itSegmentsPbID].boSelect THEN
	                #internal.panel[#PB_Configuration.itLeftSelPbID].boAborted := #internal.panel[#PB_Configuration.itLeftSelPbID].boAborted OR #EQpressL."to".boStatusAbortedSegments;
	                #internal.panel[#PB_Configuration.itLeftSelPbID].boHeld := #internal.panel[#PB_Configuration.itLeftSelPbID].boHeld OR #EQpressL."to".boStatusHeldSegments;

	                #internal.panel[#PB_Configuration.itExpandCmdPbID].boOnPos := #EQpressL."to".boPosSegmentsExp;
	                #internal.panel[#PB_Configuration.itRetractCmdPbID].boOnPos := #EQpressL."to".boPosSegmentsRet;
	                #internal.panel[#PB_Configuration.itLockCmdPbID].boOnPos := #EQpressL."to".boPosSMOLock;
	                #internal.panel[#PB_Configuration.itUnlockCmdPbID].boOnPos := #EQpressL."to".boPosSMOUnlock;

	                #internal.panel[#PB_Configuration.itExpandCmdPbID].boMoving := #EQpressL."to".boMoveSegmentsExp;
	                #internal.panel[#PB_Configuration.itRetractCmdPbID].boMoving := #EQpressL."to".boMoveSegmentsRet;
	                #internal.panel[#PB_Configuration.itLockCmdPbID].boMoving := #EQpressL."to".boMoveSMOLock;
	                #internal.panel[#PB_Configuration.itUnlockCmdPbID].boMoving := #EQpressL."to".boMoveSMOUnlock;

	                #internal.panel[#PB_Configuration.itExpandCmdPbID].boEnable := #EQpressL."to".boEnaSegmentsExp OR #internal.panel[#PB_Configuration.itExpandCmdPbID].boOnPos OR #internal.panel[#PB_Configuration.itExpandCmdPbID].boMoving;
	                #internal.panel[#PB_Configuration.itRetractCmdPbID].boEnable := #EQpressL."to".boEnaSegmentsRet OR #internal.panel[#PB_Configuration.itRetractCmdPbID].boOnPos OR #internal.panel[#PB_Configuration.itRetractCmdPbID].boMoving;
	                #internal.panel[#PB_Configuration.itLockCmdPbID].boEnable := #EQpressL."to".boEnaSMOLock OR #internal.panel[#PB_Configuration.itLockCmdPbID].boOnPos OR #internal.panel[#PB_Configuration.itLockCmdPbID].boMoving;
	                #internal.panel[#PB_Configuration.itUnlockCmdPbID].boEnable := #EQpressL."to".boEnaSMOUnlock OR #internal.panel[#PB_Configuration.itUnlockCmdPbID].boOnPos OR #internal.panel[#PB_Configuration.itUnlockCmdPbID].boMoving;

	                #EQpressL.from.boCmdSegmentsRet := #internal.panel[#PB_Configuration.itRetractCmdPbID].boCmdOn;
	                #EQpressL.from.boCmdSegmentsExp := #internal.panel[#PB_Configuration.itExpandCmdPbID].boCmdOn;
	                #EQpressL.from.boCmdSMOUnlock := #internal.panel[#PB_Configuration.itUnlockCmdPbID].boCmdOn;
	                #EQpressL.from.boCmdSMOLock := #internal.panel[#PB_Configuration.itLockCmdPbID].boCmdOn;
	            END_IF;

	            // Squeeze: manual commands
	            IF #internal.panel[#PB_Configuration.itSqueezePbID].boSelect THEN
	                #internal.panel[#PB_Configuration.itLeftSelPbID].boAborted := #internal.panel[#PB_Configuration.itLeftSelPbID].boAborted OR #EQpressL."to".boStatusAbortedSqueeze;
	                #internal.panel[#PB_Configuration.itLeftSelPbID].boHeld := #internal.panel[#PB_Configuration.itLeftSelPbID].boHeld OR #EQpressL."to".boStatusHeldSqueeze;

	                #internal.panel[#PB_Configuration.itExpandCmdPbID].boOnPos := #EQpressL."to".boPosSqueezeExp;
	                #internal.panel[#PB_Configuration.itRetractCmdPbID].boOnPos := #EQpressL."to".boPosSqueezeRet;

	                #internal.panel[#PB_Configuration.itExpandCmdPbID].boMoving := #EQpressL."to".boMoveSqueezeExp;
	                #internal.panel[#PB_Configuration.itRetractCmdPbID].boMoving := #EQpressL."to".boMoveSqueezeRet;

	                #internal.panel[#PB_Configuration.itExpandCmdPbID].boEnable := #EQpressL."to".boEnaSqueezeExp OR #internal.panel[#PB_Configuration.itExpandCmdPbID].boOnPos OR #internal.panel[#PB_Configuration.itExpandCmdPbID].boMoving;
	                #internal.panel[#PB_Configuration.itRetractCmdPbID].boEnable := #EQpressL."to".boEnaSqueezeRet OR #internal.panel[#PB_Configuration.itRetractCmdPbID].boOnPos OR #internal.panel[#PB_Configuration.itRetractCmdPbID].boMoving;

	                #EQpressL.from.boCmdSqueezeRet := #internal.panel[#PB_Configuration.itRetractCmdPbID].boCmdOn AND #internal.panel[#PB_Configuration.itLeftSelPbID].boSelect;
	                #EQpressL.from.boCmdSqueezeExp := #internal.panel[#PB_Configuration.itExpandCmdPbID].boCmdOn AND #internal.panel[#PB_Configuration.itLeftSelPbID].boSelect;
	            END_IF;
	        END_IF;

	        IF (#internal.boManSelOnPressR OR #internal.boSetupSelOnPressR OR #internal.boSetupProcActiveR) AND #internal.panel[#PB_Configuration.itRightSelPbID].boSelect THEN
	            // Enable push-buttons
	            #internal.panel[#PB_Configuration.itPressPbID].boEnable := TRUE;
	            #internal.panel[#PB_Configuration.itSegmentsPbID].boEnable := TRUE;
	            #internal.panel[#PB_Configuration.itSqueezePbID].boEnable := TRUE;

	            // Modules fault & warning
	            #internal.panel[#PB_Configuration.itPressPbID].boAborted := #EQpressR."to".boStatusAbortedEQ OR #EQpressR."to".boStatusAbortedUDMove;
	            #internal.panel[#PB_Configuration.itSegmentsPbID].boAborted := #EQpressR."to".boStatusAbortedSegments;
	            #internal.panel[#PB_Configuration.itSqueezePbID].boAborted := #EQpressR."to".boStatusAbortedSqueeze;
	            #internal.panel[#PB_Configuration.itPressPbID].boHeld := #EQpressR."to".boStatusHeldEQ OR #EQpressR."to".boStatusHeldUDMove;
	            #internal.panel[#PB_Configuration.itSegmentsPbID].boHeld := #EQpressR."to".boStatusHeldSegments;
	            #internal.panel[#PB_Configuration.itSqueezePbID].boHeld := #EQpressR."to".boStatusHeldSqueeze;

	            // Press: manual commands
	            IF #internal.panel[#PB_Configuration.itPressPbID].boSelect THEN
	                #internal.panel[#PB_Configuration.itRightSelPbID].boAborted := #internal.panel[#PB_Configuration.itRightSelPbID].boAborted OR #EQpressR."to".boStatusAbortedEQ OR #EQpressR."to".boStatusAbortedUDMove;
	                #internal.panel[#PB_Configuration.itRightSelPbID].boHeld := #internal.panel[#PB_Configuration.itRightSelPbID].boHeld OR #EQpressR."to".boStatusHeldEQ OR #EQpressR."to".boStatusHeldUDMove;

	                #internal.panel[#PB_Configuration.itUpCmdPbID].boOnPos := #EQpressR."to".boPosUDMoveUp;
	                #internal.panel[#PB_Configuration.itDownCmdPbID].boOnPos := #EQpressR."to".boPosUDMoveDown;
	                #internal.panel[#PB_Configuration.itLockCmdPbID].boOnPos := #EQpressR."to".boPosUDLock;
	                #internal.panel[#PB_Configuration.itUnlockCmdPbID].boOnPos := #EQpressR."to".boPosUDUnlock;
	                #internal.panel[#PB_Configuration.itInCmdPbID].boOnPos := #EQpressR."to".boPosSafetyBarUp;
	                #internal.panel[#PB_Configuration.itOutCmdPbID].boOnPos := #EQpressR."to".boPosSafetyBarDw;

	                #internal.panel[#PB_Configuration.itUpCmdPbID].boMoving := #EQpressR."to".boMoveUDMoveUp;
	                #internal.panel[#PB_Configuration.itDownCmdPbID].boMoving := #EQpressR."to".boMoveUDMoveDown;
	                #internal.panel[#PB_Configuration.itLockCmdPbID].boMoving := #EQpressR."to".boMoveUDLock;
	                #internal.panel[#PB_Configuration.itUnlockCmdPbID].boMoving := #EQpressR."to".boMoveUDUnlock;
	                #internal.panel[#PB_Configuration.itInCmdPbID].boMoving := #EQpressR."to".boMoveSafetyBarUp;
	                #internal.panel[#PB_Configuration.itOutCmdPbID].boMoving := #EQpressR."to".boMoveSafetyBarDw;

	                #internal.panel[#PB_Configuration.itUpCmdPbID].boEnable := #EQpressR."to".boEnaUDMoveUp OR #internal.panel[#PB_Configuration.itUpCmdPbID].boOnPos OR #internal.panel[#PB_Configuration.itUpCmdPbID].boMoving;
	                #internal.panel[#PB_Configuration.itDownCmdPbID].boEnable := #EQpressR."to".boEnaUDMoveDown OR #internal.panel[#PB_Configuration.itDownCmdPbID].boOnPos OR #internal.panel[#PB_Configuration.itDownCmdPbID].boMoving;
	                #internal.panel[#PB_Configuration.itLockCmdPbID].boEnable := #EQpressR."to".boEnaUDLock OR #internal.panel[#PB_Configuration.itLockCmdPbID].boOnPos OR #internal.panel[#PB_Configuration.itLockCmdPbID].boMoving;
	                #internal.panel[#PB_Configuration.itUnlockCmdPbID].boEnable := #EQpressR."to".boEnaUDUnlock OR #internal.panel[#PB_Configuration.itUnlockCmdPbID].boOnPos OR #internal.panel[#PB_Configuration.itUnlockCmdPbID].boMoving;
	                #internal.panel[#PB_Configuration.itInCmdPbID].boEnable := #EQpressR."to".boEnaSafetyBarUp OR #internal.panel[#PB_Configuration.itInCmdPbID].boOnPos OR #internal.panel[#PB_Configuration.itInCmdPbID].boMoving;
	                #internal.panel[#PB_Configuration.itOutCmdPbID].boEnable := #EQpressR."to".boEnaSafetyBarDw OR #internal.panel[#PB_Configuration.itOutCmdPbID].boOnPos OR #internal.panel[#PB_Configuration.itOutCmdPbID].boMoving;

	                #EQpressR.from.boCmdUDMoveDown := #internal.panel[#PB_Configuration.itDownCmdPbID].boCmdOn;
	                #EQpressR.from.boCmdUDMoveUp := #internal.panel[#PB_Configuration.itUpCmdPbID].boCmdOn;
	                #EQpressR.from.boCmdUDLock := #internal.panel[#PB_Configuration.itLockCmdPbID].boCmdOn;
	                #EQpressR.from.boCmdUDUnlock := #internal.panel[#PB_Configuration.itUnlockCmdPbID].boCmdOn;
	                #EQpressR.from.boCmdSafetyBarUp := #internal.panel[#PB_Configuration.itInCmdPbID].boCmdOn;
	                #EQpressR.from.boCmdSafetyBarDown := #internal.panel[#PB_Configuration.itOutCmdPbID].boCmdOn;
	            END_IF;

	            // Segments: manual commands
	            IF #internal.panel[#PB_Configuration.itSegmentsPbID].boSelect THEN
	                #internal.panel[#PB_Configuration.itRightSelPbID].boAborted := #internal.panel[#PB_Configuration.itRightSelPbID].boAborted OR #EQpressR."to".boStatusAbortedSegments;
	                #internal.panel[#PB_Configuration.itRightSelPbID].boHeld := #internal.panel[#PB_Configuration.itRightSelPbID].boHeld OR #EQpressR."to".boStatusHeldSegments;

	                #internal.panel[#PB_Configuration.itExpandCmdPbID].boOnPos := #EQpressR."to".boPosSegmentsExp;
	                #internal.panel[#PB_Configuration.itRetractCmdPbID].boOnPos := #EQpressR."to".boPosSegmentsRet;
	                #internal.panel[#PB_Configuration.itLockCmdPbID].boOnPos := #EQpressR."to".boPosSMOLock;
	                #internal.panel[#PB_Configuration.itUnlockCmdPbID].boOnPos := #EQpressR."to".boPosSMOUnlock;
	                #internal.panel[#PB_Configuration.itExpandCmdPbID].boMoving := #EQpressR."to".boMoveSegmentsExp;
	                #internal.panel[#PB_Configuration.itRetractCmdPbID].boMoving := #EQpressR."to".boMoveSegmentsRet;
	                #internal.panel[#PB_Configuration.itLockCmdPbID].boMoving := #EQpressR."to".boMoveSMOLock;
	                #internal.panel[#PB_Configuration.itUnlockCmdPbID].boMoving := #EQpressR."to".boMoveSMOUnlock;

	                #internal.panel[#PB_Configuration.itExpandCmdPbID].boEnable := #EQpressR."to".boEnaSegmentsExp OR #internal.panel[#PB_Configuration.itExpandCmdPbID].boOnPos OR #internal.panel[#PB_Configuration.itExpandCmdPbID].boMoving;
	                #internal.panel[#PB_Configuration.itRetractCmdPbID].boEnable := #EQpressR."to".boEnaSegmentsRet OR #internal.panel[#PB_Configuration.itRetractCmdPbID].boOnPos OR #internal.panel[#PB_Configuration.itRetractCmdPbID].boMoving;
	                #internal.panel[#PB_Configuration.itLockCmdPbID].boEnable := #EQpressR."to".boEnaSMOLock OR #internal.panel[#PB_Configuration.itLockCmdPbID].boOnPos OR #internal.panel[#PB_Configuration.itLockCmdPbID].boMoving;
	                #internal.panel[#PB_Configuration.itUnlockCmdPbID].boEnable := #EQpressL."to".boEnaSMOUnlock OR #internal.panel[#PB_Configuration.itUnlockCmdPbID].boOnPos OR #internal.panel[#PB_Configuration.itUnlockCmdPbID].boMoving;

	                #EQpressR.from.boCmdSegmentsRet := #internal.panel[#PB_Configuration.itRetractCmdPbID].boCmdOn;
	                #EQpressR.from.boCmdSegmentsExp := #internal.panel[#PB_Configuration.itExpandCmdPbID].boCmdOn;
	                #EQpressR.from.boCmdSMOUnlock := #internal.panel[#PB_Configuration.itUnlockCmdPbID].boCmdOn;
	                #EQpressR.from.boCmdSMOLock := #internal.panel[#PB_Configuration.itLockCmdPbID].boCmdOn;
	            END_IF;

	            // Squeeze: manual commands
	            IF #internal.panel[#PB_Configuration.itSqueezePbID].boSelect THEN
	                #internal.panel[#PB_Configuration.itRightSelPbID].boAborted := #internal.panel[#PB_Configuration.itRightSelPbID].boAborted OR #EQpressR."to".boStatusAbortedSqueeze;
	                #internal.panel[#PB_Configuration.itRightSelPbID].boHeld := #internal.panel[#PB_Configuration.itRightSelPbID].boHeld OR #EQpressR."to".boStatusHeldSqueeze;

	                #internal.panel[#PB_Configuration.itExpandCmdPbID].boOnPos := #EQpressR."to".boPosSqueezeExp;
	                #internal.panel[#PB_Configuration.itRetractCmdPbID].boOnPos := #EQpressR."to".boPosSqueezeRet;

	                #internal.panel[#PB_Configuration.itExpandCmdPbID].boMoving := #EQpressR."to".boMoveSqueezeExp;
	                #internal.panel[#PB_Configuration.itRetractCmdPbID].boMoving := #EQpressR."to".boMoveSqueezeRet;

	                #internal.panel[#PB_Configuration.itExpandCmdPbID].boEnable := #EQpressR."to".boEnaSqueezeExp OR #internal.panel[#PB_Configuration.itExpandCmdPbID].boOnPos OR #internal.panel[#PB_Configuration.itExpandCmdPbID].boMoving;
	                #internal.panel[#PB_Configuration.itRetractCmdPbID].boEnable := #EQpressR."to".boEnaSqueezeRet OR #internal.panel[#PB_Configuration.itRetractCmdPbID].boOnPos OR #internal.panel[#PB_Configuration.itRetractCmdPbID].boMoving;

	                #EQpressR.from.boCmdSqueezeRet := #internal.panel[#PB_Configuration.itRetractCmdPbID].boCmdOn;
	                #EQpressR.from.boCmdSqueezeExp := #internal.panel[#PB_Configuration.itExpandCmdPbID].boCmdOn;
	            END_IF;
	        END_IF;

	        IF ((#internal.boManSelOnPressL OR #internal.boSetupSelOnPressL OR #internal.boSetupProcActiveL) AND #internal.panel[#PB_Configuration.itLeftSelPbID].boSelect) AND
	            ((#internal.boManSelOnPressR OR #internal.boSetupSelOnPressR OR #internal.boSetupProcActiveR) AND #internal.panel[#PB_Configuration.itRightSelPbID].boSelect) THEN
	            // Enable push-buttons
	            #internal.panel[#PB_Configuration.itPressPbID].boEnable := TRUE;
	            #internal.panel[#PB_Configuration.itSegmentsPbID].boEnable := TRUE;
	            #internal.panel[#PB_Configuration.itSqueezePbID].boEnable := TRUE;

	            // Modules fault & warning
	            #internal.panel[#PB_Configuration.itPressPbID].boAborted := #EQpressL."to".boStatusAbortedEQ OR #EQpressL."to".boStatusAbortedUDMove OR #EQpressR."to".boStatusAbortedEQ OR #EQpressR."to".boStatusAbortedUDMove;
	            #internal.panel[#PB_Configuration.itSegmentsPbID].boAborted := #EQpressL."to".boStatusAbortedSegments OR #EQpressR."to".boStatusAbortedSegments;
	            #internal.panel[#PB_Configuration.itSqueezePbID].boAborted := #EQpressL."to".boStatusAbortedSqueeze OR #EQpressR."to".boStatusAbortedSqueeze;
	            #internal.panel[#PB_Configuration.itPressPbID].boHeld := #EQpressL."to".boStatusHeldEQ OR #EQpressL."to".boStatusHeldUDMove OR #EQpressR."to".boStatusHeldEQ OR #EQpressR."to".boStatusHeldUDMove;
	            #internal.panel[#PB_Configuration.itSegmentsPbID].boHeld := #EQpressL."to".boStatusHeldSegments OR #EQpressR."to".boStatusHeldSegments;
	            #internal.panel[#PB_Configuration.itSqueezePbID].boHeld := #EQpressL."to".boStatusHeldSqueeze OR #EQpressR."to".boStatusHeldSqueeze;

	            // Press: manual commands
	            IF #internal.panel[#PB_Configuration.itPressPbID].boSelect THEN
	                #internal.panel[#PB_Configuration.itUpCmdPbID].boOnPos := #EQpressL."to".boPosUDMoveUp AND #EQpressR."to".boPosUDMoveUp;
	                #internal.panel[#PB_Configuration.itDownCmdPbID].boOnPos := #EQpressL."to".boPosUDMoveDown AND #EQpressR."to".boPosUDMoveDown;
	                #internal.panel[#PB_Configuration.itLockCmdPbID].boOnPos := #EQpressL."to".boPosUDLock AND #EQpressR."to".boPosUDLock;
	                #internal.panel[#PB_Configuration.itUnlockCmdPbID].boOnPos := #EQpressL."to".boPosUDUnlock AND #EQpressR."to".boPosUDUnlock;

	                #internal.panel[#PB_Configuration.itUpCmdPbID].boMoving := #EQpressL."to".boMoveUDMoveUp OR #EQpressR."to".boMoveUDMoveUp;
	                #internal.panel[#PB_Configuration.itDownCmdPbID].boMoving := #EQpressL."to".boMoveUDMoveDown OR #EQpressR."to".boMoveUDMoveDown;
	                #internal.panel[#PB_Configuration.itLockCmdPbID].boMoving := #EQpressL."to".boMoveUDLock OR #EQpressR."to".boMoveUDLock;
	                #internal.panel[#PB_Configuration.itUnlockCmdPbID].boMoving := #EQpressL."to".boMoveUDUnlock OR #EQpressR."to".boMoveUDUnlock;

	                #internal.panel[#PB_Configuration.itUpCmdPbID].boEnable := #EQpressL."to".boEnaUDMoveUp OR #EQpressR."to".boEnaUDMoveUp OR #internal.panel[#PB_Configuration.itUpCmdPbID].boOnPos OR #internal.panel[#PB_Configuration.itUpCmdPbID].boMoving;
	                #internal.panel[#PB_Configuration.itDownCmdPbID].boEnable := #EQpressL."to".boEnaUDMoveDown OR #EQpressR."to".boEnaUDMoveDown OR #internal.panel[#PB_Configuration.itDownCmdPbID].boOnPos OR #internal.panel[#PB_Configuration.itDownCmdPbID].boMoving;
	                #internal.panel[#PB_Configuration.itLockCmdPbID].boEnable := #EQpressL."to".boEnaUDLock OR #EQpressR."to".boEnaUDLock OR #internal.panel[#PB_Configuration.itLockCmdPbID].boOnPos OR #internal.panel[#PB_Configuration.itLockCmdPbID].boMoving;
	                #internal.panel[#PB_Configuration.itUnlockCmdPbID].boEnable := #EQpressL."to".boEnaUDUnlock OR #EQpressR."to".boEnaUDUnlock OR #internal.panel[#PB_Configuration.itUnlockCmdPbID].boOnPos OR #internal.panel[#PB_Configuration.itUnlockCmdPbID].boMoving;
	            END_IF;

	            // Segments: manual commands
	            IF #internal.panel[#PB_Configuration.itSegmentsPbID].boSelect THEN
	                #internal.panel[#PB_Configuration.itExpandCmdPbID].boOnPos := #EQpressL."to".boPosSegmentsExp AND #EQpressR."to".boPosSegmentsExp;
	                #internal.panel[#PB_Configuration.itRetractCmdPbID].boOnPos := #EQpressL."to".boPosSegmentsRet AND #EQpressR."to".boPosSegmentsRet;
	                #internal.panel[#PB_Configuration.itLockCmdPbID].boOnPos := #EQpressL."to".boPosSMOLock AND #EQpressR."to".boPosSMOLock;
	                #internal.panel[#PB_Configuration.itUnlockCmdPbID].boOnPos := #EQpressL."to".boPosSMOUnlock AND #EQpressR."to".boPosSMOUnlock;

	                #internal.panel[#PB_Configuration.itExpandCmdPbID].boMoving := #EQpressL."to".boMoveSegmentsExp OR #EQpressR."to".boMoveSegmentsExp;
	                #internal.panel[#PB_Configuration.itRetractCmdPbID].boMoving := #EQpressL."to".boMoveSegmentsRet OR #EQpressR."to".boMoveSegmentsRet;
	                #internal.panel[#PB_Configuration.itLockCmdPbID].boMoving := #EQpressL."to".boMoveSMOLock OR #EQpressL."to".boMoveSMOLock;
	                #internal.panel[#PB_Configuration.itUnlockCmdPbID].boMoving := #EQpressL."to".boMoveSMOUnlock OR #EQpressR."to".boMoveSMOUnlock;

	                #internal.panel[#PB_Configuration.itExpandCmdPbID].boEnable := #EQpressL."to".boEnaSegmentsExp OR #EQpressR."to".boEnaSegmentsExp OR #internal.panel[#PB_Configuration.itExpandCmdPbID].boOnPos OR #internal.panel[#PB_Configuration.itExpandCmdPbID].boMoving;
	                #internal.panel[#PB_Configuration.itRetractCmdPbID].boEnable := #EQpressL."to".boEnaSegmentsRet OR #EQpressR."to".boEnaSegmentsRet OR #internal.panel[#PB_Configuration.itRetractCmdPbID].boOnPos OR #internal.panel[#PB_Configuration.itRetractCmdPbID].boMoving;
	                #internal.panel[#PB_Configuration.itLockCmdPbID].boEnable := #EQpressL."to".boEnaSMOLock OR #EQpressR."to".boEnaSMOLock OR #internal.panel[#PB_Configuration.itLockCmdPbID].boOnPos OR #internal.panel[#PB_Configuration.itLockCmdPbID].boMoving;
	                #internal.panel[#PB_Configuration.itUnlockCmdPbID].boEnable := #EQpressL."to".boEnaSMOUnlock OR #EQpressR."to".boEnaSMOUnlock OR #internal.panel[#PB_Configuration.itUnlockCmdPbID].boOnPos OR #internal.panel[#PB_Configuration.itUnlockCmdPbID].boMoving;
	            END_IF;

	            // Squeeze: manual commands
	            IF #internal.panel[#PB_Configuration.itSqueezePbID].boSelect THEN
	                #internal.panel[#PB_Configuration.itExpandCmdPbID].boOnPos := #EQpressL."to".boPosSqueezeExp AND #EQpressR."to".boPosSqueezeExp;
	                #internal.panel[#PB_Configuration.itRetractCmdPbID].boOnPos := #EQpressL."to".boPosSqueezeRet AND #EQpressR."to".boPosSqueezeRet;

	                #internal.panel[#PB_Configuration.itExpandCmdPbID].boMoving := #EQpressL."to".boMoveSqueezeExp OR #EQpressR."to".boMoveSqueezeExp;
	                #internal.panel[#PB_Configuration.itRetractCmdPbID].boMoving := #EQpressL."to".boMoveSqueezeRet OR #EQpressR."to".boMoveSqueezeRet;

	                #internal.panel[#PB_Configuration.itExpandCmdPbID].boEnable := #EQpressL."to".boEnaSqueezeExp OR #EQpressR."to".boEnaSqueezeExp OR #internal.panel[#PB_Configuration.itExpandCmdPbID].boOnPos OR #internal.panel[#PB_Configuration.itExpandCmdPbID].boMoving;
	                #internal.panel[#PB_Configuration.itRetractCmdPbID].boEnable := #EQpressL."to".boEnaSqueezeRet OR #EQpressR."to".boEnaSqueezeRet OR #internal.panel[#PB_Configuration.itRetractCmdPbID].boOnPos OR #internal.panel[#PB_Configuration.itRetractCmdPbID].boMoving;
	            END_IF;
	        END_IF;
	    END_REGION

	    REGION CENTER-MECH
	        IF (#internal.boManSelOnPressL OR #internal.boSetupSelOnPressL OR #internal.boSetupProcActiveL) AND #internal.panel[#PB_Configuration.itLeftSelPbID].boSelect THEN
	            // Enable push-buttons
	            #internal.panel[#PB_Configuration.itTopRingPbID].boEnable := TRUE;
	            #internal.panel[#PB_Configuration.itBotRingPbID].boEnable := TRUE;
	            #internal.panel[#PB_Configuration.itBeadRingPbID].boEnable := TRUE;

	            // Modules fault & warning
	            #internal.panel[#PB_Configuration.itTopRingPbID].boAborted := #EQcenterMechL."to".boStatusAbortedEQ OR #EQcenterMechL."to".boStatusAbortedTCRing;
	            #internal.panel[#PB_Configuration.itBotRingPbID].boAborted := #EQcenterMechL."to".boStatusAbortedBCRing;
	            #internal.panel[#PB_Configuration.itBeadRingPbID].boAborted := #EQcenterMechL."to".boStatusAbortedBeadRing;
	            #internal.panel[#PB_Configuration.itTopRingPbID].boHeld := #EQcenterMechL."to".boStatusHeldEQ OR #EQcenterMechL."to".boStatusHeldTCRing;
	            #internal.panel[#PB_Configuration.itBotRingPbID].boHeld := #EQcenterMechL."to".boStatusHeldBCRing;
	            #internal.panel[#PB_Configuration.itBeadRingPbID].boHeld := #EQcenterMechL."to".boStatusHeldBeadRing;

	            // Top-Rings: manual commands
	            IF #internal.panel[#PB_Configuration.itTopRingPbID].boSelect THEN
	                #internal.panel[#PB_Configuration.itLeftSelPbID].boAborted := #EQcenterMechL."to".boStatusAbortedEQ OR #EQcenterMechL."to".boStatusAbortedTCRing;
	                #internal.panel[#PB_Configuration.itLeftSelPbID].boHeld := #EQcenterMechL."to".boStatusHeldEQ OR #EQcenterMechL."to".boStatusHeldTCRing;

	                #internal.panel[#PB_Configuration.itUpCmdPbID].boOnPos := #EQcenterMechL."to".boPosTCRingUp;
	                #internal.panel[#PB_Configuration.itDownCmdPbID].boOnPos := #EQcenterMechL."to".boPosTCRingDown;

	                #internal.panel[#PB_Configuration.itUpCmdPbID].boMoving := #EQcenterMechL."to".boMoveTCRingUp;
	                #internal.panel[#PB_Configuration.itDownCmdPbID].boMoving := #EQcenterMechL."to".boMoveTCRingDown;

	                #internal.panel[#PB_Configuration.itUpCmdPbID].boEnable := #EQcenterMechL."to".boEnaTCRingUp OR #internal.panel[#PB_Configuration.itUpCmdPbID].boOnPos OR #internal.panel[#PB_Configuration.itUpCmdPbID].boMoving;
	                #internal.panel[#PB_Configuration.itDownCmdPbID].boEnable := #EQcenterMechL."to".boEnaTCRingDown OR #internal.panel[#PB_Configuration.itDownCmdPbID].boOnPos OR #internal.panel[#PB_Configuration.itDownCmdPbID].boMoving;

	                #EQcenterMechL.from.boCmdTCRingDown := #internal.panel[#PB_Configuration.itDownCmdPbID].boCmdOn;
	                #EQcenterMechL.from.boCmdTCRingUp := #internal.panel[#PB_Configuration.itUpCmdPbID].boCmdOn;
	            END_IF;

	            // Bottom-Rings: manual commands
	            IF #internal.panel[#PB_Configuration.itBotRingPbID].boSelect THEN
	                #internal.panel[#PB_Configuration.itLeftSelPbID].boAborted := #EQcenterMechL."to".boStatusAbortedBCRing;
	                #internal.panel[#PB_Configuration.itLeftSelPbID].boHeld := #EQcenterMechL."to".boStatusHeldBCRing;

	                #internal.panel[#PB_Configuration.itUpCmdPbID].boOnPos := #EQcenterMechL."to".boPosBCRingUp;
	                #internal.panel[#PB_Configuration.itDownCmdPbID].boOnPos := #EQcenterMechL."to".boPosBCRingDown;
	                #internal.panel[#PB_Configuration.itLockCmdPbID].boOnPos := #EQcenterMechL."to".boPosBCRingLock;
	                #internal.panel[#PB_Configuration.itUnlockCmdPbID].boOnPos := #EQcenterMechL."to".boPosBCRingUnlock;

	                #internal.panel[#PB_Configuration.itUpCmdPbID].boMoving := #EQcenterMechL."to".boMoveBCRingUp;
	                #internal.panel[#PB_Configuration.itDownCmdPbID].boMoving := #EQcenterMechL."to".boMoveBCRingDown;
	                #internal.panel[#PB_Configuration.itLockCmdPbID].boMoving := #EQcenterMechL."to".boMoveBCRingLock;
	                #internal.panel[#PB_Configuration.itUnlockCmdPbID].boMoving := #EQcenterMechL."to".boMoveBCRingUnlock;

	                #internal.panel[#PB_Configuration.itUpCmdPbID].boEnable := #EQcenterMechL."to".boEnaBCRingUp OR #internal.panel[#PB_Configuration.itUpCmdPbID].boOnPos OR #internal.panel[#PB_Configuration.itUpCmdPbID].boMoving;
	                #internal.panel[#PB_Configuration.itDownCmdPbID].boEnable := #EQcenterMechL."to".boEnaBCRingDown OR #internal.panel[#PB_Configuration.itDownCmdPbID].boOnPos OR #internal.panel[#PB_Configuration.itDownCmdPbID].boMoving;
	                #internal.panel[#PB_Configuration.itLockCmdPbID].boEnable := #EQcenterMechL."to".boEnaBCRingLock OR #internal.panel[#PB_Configuration.itLockCmdPbID].boOnPos OR #internal.panel[#PB_Configuration.itLockCmdPbID].boMoving;
	                #internal.panel[#PB_Configuration.itUnlockCmdPbID].boEnable := #EQcenterMechL."to".boEnaBCRingUnlock OR #internal.panel[#PB_Configuration.itUnlockCmdPbID].boOnPos OR #internal.panel[#PB_Configuration.itUnlockCmdPbID].boMoving;

	                #EQcenterMechL.from.boCmdBCRingDown := #internal.panel[#PB_Configuration.itDownCmdPbID].boCmdOn;
	                #EQcenterMechL.from.boCmdBCRingUp := #internal.panel[#PB_Configuration.itUpCmdPbID].boCmdOn;
	                #EQcenterMechL.from.boCmdBCRingLock := #internal.panel[#PB_Configuration.itLockCmdPbID].boCmdOn;
	                #EQcenterMechL.from.boCmdBCRingUnlock := #internal.panel[#PB_Configuration.itUnlockCmdPbID].boCmdOn;
	            END_IF;

	            // Bead-Rings: manual commands
	            IF #internal.panel[#PB_Configuration.itBeadRingPbID].boSelect THEN
	                #internal.panel[#PB_Configuration.itLeftSelPbID].boAborted := #EQcenterMechL."to".boStatusAbortedBeadRing;
	                #internal.panel[#PB_Configuration.itLeftSelPbID].boHeld := #EQcenterMechL."to".boStatusHeldBeadRing;

	                #internal.panel[#PB_Configuration.itUpCmdPbID].boOnPos := #EQcenterMechL."to".boPosBeadRingUp;
	                #internal.panel[#PB_Configuration.itDownCmdPbID].boOnPos := #EQcenterMechL."to".boPosBeadRingDown;

	                #internal.panel[#PB_Configuration.itUpCmdPbID].boMoving := #EQcenterMechL."to".boMoveBeadRingUp;
	                #internal.panel[#PB_Configuration.itDownCmdPbID].boMoving := #EQcenterMechL."to".boMoveBeadRingDown;

	                #internal.panel[#PB_Configuration.itUpCmdPbID].boEnable := #EQcenterMechL."to".boEnaBeadRingUp OR #internal.panel[#PB_Configuration.itUpCmdPbID].boOnPos OR #internal.panel[#PB_Configuration.itUpCmdPbID].boMoving;
	                #internal.panel[#PB_Configuration.itDownCmdPbID].boEnable := #EQcenterMechL."to".boEnaBeadRingDown OR #internal.panel[#PB_Configuration.itDownCmdPbID].boOnPos OR #internal.panel[#PB_Configuration.itDownCmdPbID].boMoving;

	                #EQcenterMechL.from.boCmdBeadRingDown := #internal.panel[#PB_Configuration.itDownCmdPbID].boCmdOn;
	                #EQcenterMechL.from.boCmdBeadRingUp := #internal.panel[#PB_Configuration.itUpCmdPbID].boCmdOn;
	            END_IF;
	        END_IF;

	        IF (#internal.boManSelOnPressR OR #internal.boSetupSelOnPressR OR #internal.boSetupProcActiveR) AND #internal.panel[#PB_Configuration.itRightSelPbID].boSelect THEN
	            // Enable push-buttons
	            #internal.panel[#PB_Configuration.itTopRingPbID].boEnable := TRUE;
	            #internal.panel[#PB_Configuration.itBotRingPbID].boEnable := TRUE;
	            #internal.panel[#PB_Configuration.itBeadRingPbID].boEnable := TRUE;

	            // Modules fault & warning
	            #internal.panel[#PB_Configuration.itTopRingPbID].boAborted := #EQcenterMechR."to".boStatusAbortedEQ OR #EQcenterMechR."to".boStatusAbortedTCRing;
	            #internal.panel[#PB_Configuration.itBotRingPbID].boAborted := #EQcenterMechR."to".boStatusAbortedBCRing;
	            #internal.panel[#PB_Configuration.itBeadRingPbID].boAborted := #EQcenterMechR."to".boStatusAbortedBeadRing;
	            #internal.panel[#PB_Configuration.itTopRingPbID].boHeld := #EQcenterMechR."to".boStatusHeldEQ OR #EQcenterMechR."to".boStatusHeldTCRing;
	            #internal.panel[#PB_Configuration.itBotRingPbID].boHeld := #EQcenterMechR."to".boStatusHeldBCRing;
	            #internal.panel[#PB_Configuration.itBeadRingPbID].boHeld := #EQcenterMechR."to".boStatusHeldBeadRing;

	            // Top-Rings: manual commands
	            IF #internal.panel[#PB_Configuration.itTopRingPbID].boSelect THEN
	                #internal.panel[#PB_Configuration.itRightSelPbID].boAborted := #EQcenterMechR."to".boStatusAbortedEQ OR #EQcenterMechR."to".boStatusAbortedTCRing;
	                #internal.panel[#PB_Configuration.itRightSelPbID].boHeld := #EQcenterMechR."to".boStatusHeldEQ OR #EQcenterMechR."to".boStatusHeldTCRing;

	                #internal.panel[#PB_Configuration.itUpCmdPbID].boOnPos := #EQcenterMechR."to".boPosTCRingUp;
	                #internal.panel[#PB_Configuration.itDownCmdPbID].boOnPos := #EQcenterMechR."to".boPosTCRingDown;

	                #internal.panel[#PB_Configuration.itUpCmdPbID].boMoving := #EQcenterMechR."to".boMoveTCRingUp;
	                #internal.panel[#PB_Configuration.itDownCmdPbID].boMoving := #EQcenterMechR."to".boMoveTCRingDown;

	                #internal.panel[#PB_Configuration.itUpCmdPbID].boEnable := #EQcenterMechR."to".boEnaTCRingUp OR #internal.panel[#PB_Configuration.itUpCmdPbID].boOnPos OR #internal.panel[#PB_Configuration.itUpCmdPbID].boMoving;
	                #internal.panel[#PB_Configuration.itDownCmdPbID].boEnable := #EQcenterMechR."to".boEnaTCRingDown OR #internal.panel[#PB_Configuration.itDownCmdPbID].boOnPos OR #internal.panel[#PB_Configuration.itDownCmdPbID].boMoving;

	                #EQcenterMechR.from.boCmdTCRingDown := #internal.panel[#PB_Configuration.itDownCmdPbID].boCmdOn;
	                #EQcenterMechR.from.boCmdTCRingUp := #internal.panel[#PB_Configuration.itUpCmdPbID].boCmdOn;
	            END_IF;

	            // Bottom-Rings: manual commands
	            IF #internal.panel[#PB_Configuration.itBotRingPbID].boSelect THEN
	                #internal.panel[#PB_Configuration.itRightSelPbID].boAborted := #EQcenterMechR."to".boStatusAbortedBCRing;
	                #internal.panel[#PB_Configuration.itRightSelPbID].boHeld := #EQcenterMechR."to".boStatusHeldBCRing;

	                #internal.panel[#PB_Configuration.itUpCmdPbID].boOnPos := #EQcenterMechR."to".boPosBCRingUp;
	                #internal.panel[#PB_Configuration.itDownCmdPbID].boOnPos := #EQcenterMechR."to".boPosBCRingDown;
	                #internal.panel[#PB_Configuration.itLockCmdPbID].boOnPos := #EQcenterMechR."to".boPosBCRingLock;
	                #internal.panel[#PB_Configuration.itUnlockCmdPbID].boOnPos := #EQcenterMechR."to".boPosBCRingUnlock;

	                #internal.panel[#PB_Configuration.itUpCmdPbID].boMoving := #EQcenterMechR."to".boMoveBCRingUp;
	                #internal.panel[#PB_Configuration.itDownCmdPbID].boMoving := #EQcenterMechR."to".boMoveBCRingDown;
	                #internal.panel[#PB_Configuration.itLockCmdPbID].boMoving := #EQcenterMechR."to".boMoveBCRingLock;
	                #internal.panel[#PB_Configuration.itUnlockCmdPbID].boMoving := #EQcenterMechR."to".boMoveBCRingUnlock;

	                #internal.panel[#PB_Configuration.itUpCmdPbID].boEnable := #EQcenterMechR."to".boEnaBCRingUp OR #internal.panel[#PB_Configuration.itUpCmdPbID].boOnPos OR #internal.panel[#PB_Configuration.itUpCmdPbID].boMoving;
	                #internal.panel[#PB_Configuration.itDownCmdPbID].boEnable := #EQcenterMechR."to".boEnaBCRingDown OR #internal.panel[#PB_Configuration.itDownCmdPbID].boOnPos OR #internal.panel[#PB_Configuration.itDownCmdPbID].boMoving;
	                #internal.panel[#PB_Configuration.itLockCmdPbID].boEnable := #EQcenterMechR."to".boEnaBCRingLock OR #internal.panel[#PB_Configuration.itLockCmdPbID].boOnPos OR #internal.panel[#PB_Configuration.itLockCmdPbID].boMoving;
	                #internal.panel[#PB_Configuration.itUnlockCmdPbID].boEnable := #EQcenterMechR."to".boEnaBCRingUnlock OR #internal.panel[#PB_Configuration.itUnlockCmdPbID].boOnPos OR #internal.panel[#PB_Configuration.itUnlockCmdPbID].boMoving;

	                #EQcenterMechR.from.boCmdBCRingDown := #internal.panel[#PB_Configuration.itDownCmdPbID].boCmdOn;
	                #EQcenterMechR.from.boCmdBCRingUp := #internal.panel[#PB_Configuration.itUpCmdPbID].boCmdOn;
	                #EQcenterMechR.from.boCmdBCRingLock := #internal.panel[#PB_Configuration.itLockCmdPbID].boCmdOn;
	                #EQcenterMechR.from.boCmdBCRingUnlock := #internal.panel[#PB_Configuration.itUnlockCmdPbID].boCmdOn;
	            END_IF;

	            // Bead-Rings: manual commands
	            IF #internal.panel[#PB_Configuration.itBeadRingPbID].boSelect THEN
	                #internal.panel[#PB_Configuration.itRightSelPbID].boAborted := #EQcenterMechR."to".boStatusAbortedBeadRing;
	                #internal.panel[#PB_Configuration.itRightSelPbID].boHeld := #EQcenterMechR."to".boStatusHeldBeadRing;

	                #internal.panel[#PB_Configuration.itUpCmdPbID].boOnPos := #EQcenterMechR."to".boPosBeadRingUp;
	                #internal.panel[#PB_Configuration.itDownCmdPbID].boOnPos := #EQcenterMechR."to".boPosBeadRingDown;

	                #internal.panel[#PB_Configuration.itUpCmdPbID].boMoving := #EQcenterMechR."to".boMoveBeadRingUp;
	                #internal.panel[#PB_Configuration.itDownCmdPbID].boMoving := #EQcenterMechR."to".boMoveBeadRingDown;

	                #internal.panel[#PB_Configuration.itUpCmdPbID].boEnable := #EQcenterMechR."to".boEnaBeadRingUp OR #internal.panel[#PB_Configuration.itUpCmdPbID].boOnPos OR #internal.panel[#PB_Configuration.itUpCmdPbID].boMoving;
	                #internal.panel[#PB_Configuration.itDownCmdPbID].boEnable := #EQcenterMechR."to".boEnaBeadRingDown OR #internal.panel[#PB_Configuration.itDownCmdPbID].boOnPos OR #internal.panel[#PB_Configuration.itDownCmdPbID].boMoving;

	                #EQcenterMechR.from.boCmdBeadRingDown := #internal.panel[#PB_Configuration.itDownCmdPbID].boCmdOn AND #internal.panel[#PB_Configuration.itRightSelPbID].boSelect;
	                #EQcenterMechR.from.boCmdBeadRingUp := #internal.panel[#PB_Configuration.itUpCmdPbID].boCmdOn AND #internal.panel[#PB_Configuration.itRightSelPbID].boSelect;
	            END_IF;
	        END_IF;

	        IF ((#internal.boManSelOnPressL OR #internal.boSetupSelOnPressL OR #internal.boSetupProcActiveL) AND #internal.panel[#PB_Configuration.itLeftSelPbID].boSelect) AND
	            ((#internal.boManSelOnPressR OR #internal.boSetupSelOnPressR OR #internal.boSetupProcActiveR) AND #internal.panel[#PB_Configuration.itRightSelPbID].boSelect) THEN
	            // Enable push-buttons
	            #internal.panel[#PB_Configuration.itTopRingPbID].boEnable := TRUE;
	            #internal.panel[#PB_Configuration.itBotRingPbID].boEnable := TRUE;
	            #internal.panel[#PB_Configuration.itBeadRingPbID].boEnable := TRUE;

	            // Modules fault & warning
	            #internal.panel[#PB_Configuration.itTopRingPbID].boAborted := #EQcenterMechL."to".boStatusAbortedEQ OR #EQcenterMechL."to".boStatusAbortedTCRing OR #EQcenterMechR."to".boStatusAbortedEQ OR #EQcenterMechR."to".boStatusAbortedTCRing;
	            #internal.panel[#PB_Configuration.itBotRingPbID].boAborted := #EQcenterMechL."to".boStatusAbortedBCRing OR #EQcenterMechR."to".boStatusAbortedBCRing;
	            #internal.panel[#PB_Configuration.itBeadRingPbID].boAborted := #EQcenterMechL."to".boStatusAbortedBeadRing OR #EQcenterMechR."to".boStatusAbortedBeadRing;
	            #internal.panel[#PB_Configuration.itTopRingPbID].boHeld := #EQcenterMechL."to".boStatusHeldEQ OR #EQcenterMechL."to".boStatusHeldTCRing OR #EQcenterMechR."to".boStatusHeldEQ OR #EQcenterMechR."to".boStatusHeldTCRing;
	            #internal.panel[#PB_Configuration.itBotRingPbID].boHeld := #EQcenterMechL."to".boStatusHeldBCRing OR #EQcenterMechR."to".boStatusHeldBCRing;
	            #internal.panel[#PB_Configuration.itBeadRingPbID].boHeld := #EQcenterMechL."to".boStatusHeldBeadRing OR #EQcenterMechR."to".boStatusHeldBeadRing;

	            // Top-Rings: manual commands
	            IF #internal.panel[#PB_Configuration.itTopRingPbID].boSelect THEN
	                #internal.panel[#PB_Configuration.itUpCmdPbID].boOnPos := #EQcenterMechL."to".boPosTCRingUp AND #EQcenterMechR."to".boPosTCRingUp;
	                #internal.panel[#PB_Configuration.itDownCmdPbID].boOnPos := #EQcenterMechL."to".boPosTCRingDown AND #EQcenterMechR."to".boPosTCRingDown;

	                #internal.panel[#PB_Configuration.itUpCmdPbID].boMoving := #EQcenterMechL."to".boMoveTCRingUp OR #EQcenterMechR."to".boMoveTCRingUp;
	                #internal.panel[#PB_Configuration.itDownCmdPbID].boMoving := #EQcenterMechL."to".boMoveTCRingDown OR #EQcenterMechR."to".boMoveTCRingDown;

	                #internal.panel[#PB_Configuration.itUpCmdPbID].boEnable := #EQcenterMechL."to".boEnaTCRingUp OR #EQcenterMechR."to".boEnaTCRingUp OR #internal.panel[#PB_Configuration.itUpCmdPbID].boOnPos OR #internal.panel[#PB_Configuration.itUpCmdPbID].boMoving;
	                #internal.panel[#PB_Configuration.itDownCmdPbID].boEnable := #EQcenterMechL."to".boEnaTCRingDown OR #EQcenterMechR."to".boEnaTCRingDown OR #internal.panel[#PB_Configuration.itDownCmdPbID].boOnPos OR #internal.panel[#PB_Configuration.itDownCmdPbID].boMoving;
	            END_IF;

	            // Bottom-Rings: manual commands
	            IF #internal.panel[#PB_Configuration.itBotRingPbID].boSelect THEN
	                #internal.panel[#PB_Configuration.itUpCmdPbID].boOnPos := #EQcenterMechL."to".boPosBCRingUp AND #EQcenterMechR."to".boPosBCRingUp;
	                #internal.panel[#PB_Configuration.itDownCmdPbID].boOnPos := #EQcenterMechL."to".boPosBCRingDown AND #EQcenterMechR."to".boPosBCRingDown;
	                #internal.panel[#PB_Configuration.itLockCmdPbID].boOnPos := #EQcenterMechL."to".boPosBCRingLock AND #EQcenterMechR."to".boPosBCRingLock;
	                #internal.panel[#PB_Configuration.itUnlockCmdPbID].boOnPos := #EQcenterMechL."to".boPosBCRingUnlock AND #EQcenterMechR."to".boPosBCRingUnlock;

	                #internal.panel[#PB_Configuration.itUpCmdPbID].boMoving := #EQcenterMechL."to".boMoveBCRingUp OR #EQcenterMechR."to".boMoveBCRingUp;
	                #internal.panel[#PB_Configuration.itDownCmdPbID].boMoving := #EQcenterMechL."to".boMoveBCRingDown OR #EQcenterMechR."to".boMoveBCRingDown;
	                #internal.panel[#PB_Configuration.itLockCmdPbID].boMoving := #EQcenterMechL."to".boMoveBCRingLock OR #EQcenterMechR."to".boMoveBCRingLock;
	                #internal.panel[#PB_Configuration.itUnlockCmdPbID].boMoving := #EQcenterMechL."to".boMoveBCRingUnlock OR #EQcenterMechR."to".boMoveBCRingUnlock;

	                #internal.panel[#PB_Configuration.itUpCmdPbID].boEnable := #EQcenterMechL."to".boEnaBCRingUp OR #EQcenterMechR."to".boEnaBCRingUp OR #internal.panel[#PB_Configuration.itUpCmdPbID].boOnPos OR #internal.panel[#PB_Configuration.itUpCmdPbID].boMoving;
	                #internal.panel[#PB_Configuration.itDownCmdPbID].boEnable := #EQcenterMechL."to".boEnaBCRingDown OR #EQcenterMechR."to".boEnaBCRingDown OR #internal.panel[#PB_Configuration.itDownCmdPbID].boOnPos OR #internal.panel[#PB_Configuration.itDownCmdPbID].boMoving;
	                #internal.panel[#PB_Configuration.itLockCmdPbID].boEnable := #EQcenterMechL."to".boEnaBCRingLock OR #EQcenterMechR."to".boEnaBCRingLock OR #internal.panel[#PB_Configuration.itLockCmdPbID].boOnPos OR #internal.panel[#PB_Configuration.itLockCmdPbID].boMoving;
	                #internal.panel[#PB_Configuration.itUnlockCmdPbID].boEnable := #EQcenterMechL."to".boEnaBCRingUnlock OR #EQcenterMechR."to".boEnaBCRingUnlock OR #internal.panel[#PB_Configuration.itUnlockCmdPbID].boOnPos OR #internal.panel[#PB_Configuration.itUnlockCmdPbID].boMoving;
	            END_IF;

	            // Bead-Rings: manual commands
	            IF #internal.panel[#PB_Configuration.itBeadRingPbID].boSelect THEN
	                #internal.panel[#PB_Configuration.itUpCmdPbID].boOnPos := #EQcenterMechL."to".boPosBeadRingUp AND #EQcenterMechR."to".boPosBeadRingUp;
	                #internal.panel[#PB_Configuration.itDownCmdPbID].boOnPos := #EQcenterMechL."to".boPosBeadRingDown AND #EQcenterMechR."to".boPosBeadRingDown;

	                #internal.panel[#PB_Configuration.itUpCmdPbID].boMoving := #EQcenterMechL."to".boMoveBeadRingUp OR #EQcenterMechR."to".boMoveBeadRingUp;
	                #internal.panel[#PB_Configuration.itDownCmdPbID].boMoving := #EQcenterMechL."to".boMoveBeadRingDown OR #EQcenterMechR."to".boMoveBeadRingDown;

	                #internal.panel[#PB_Configuration.itUpCmdPbID].boEnable := #EQcenterMechL."to".boEnaBeadRingUp OR #EQcenterMechR."to".boEnaBeadRingUp OR #internal.panel[#PB_Configuration.itUpCmdPbID].boOnPos OR #internal.panel[#PB_Configuration.itUpCmdPbID].boMoving;
	                #internal.panel[#PB_Configuration.itDownCmdPbID].boEnable := #EQcenterMechL."to".boEnaBeadRingDown OR #EQcenterMechR."to".boEnaBeadRingDown OR #internal.panel[#PB_Configuration.itDownCmdPbID].boOnPos OR #internal.panel[#PB_Configuration.itDownCmdPbID].boMoving;
	            END_IF;
	        END_IF;
	    END_REGION

	    REGION HEATING (INTERNAL & EXTERNAL)
	        IF (#internal.boManSelOnHeatingL OR #internal.boSetupSelOnHeatingL OR #internal.boSetupProcActiveL) AND #internal.panel[#PB_Configuration.itLeftSelPbID].boSelect THEN
	            // Enable push-buttons
	            #internal.panel[#PB_Configuration.itShapingPbID].boEnable := TRUE;
	            #internal.panel[#PB_Configuration.itDrainPbID].boEnable := TRUE;
	            #internal.panel[#PB_Configuration.itVacuumPbID].boEnable := TRUE;

	            // Modules fault & warning
	            #internal.panel[#PB_Configuration.itShapingPbID].boAborted := #EQintHeatL."to".boStatusAbortedEQ OR #EQintHeatL."to".boStatusAbortedShape;
	            #internal.panel[#PB_Configuration.itDrainPbID].boAborted := #EQintHeatL."to".boStatusAbortedDrain;
	            #internal.panel[#PB_Configuration.itVacuumPbID].boAborted := #EQintHeatL."to".boStatusAbortedVacuum;
	            #internal.panel[#PB_Configuration.itShapingPbID].boHeld := #EQintHeatL."to".boStatusHeldEQ OR #EQintHeatL."to".boStatusHeldShape;
	            #internal.panel[#PB_Configuration.itDrainPbID].boHeld := #EQintHeatL."to".boStatusHeldDrain;
	            #internal.panel[#PB_Configuration.itVacuumPbID].boHeld := #EQintHeatL."to".boStatusHeldVacuum;

	            // Shaping: manual commands
	            IF #internal.panel[#PB_Configuration.itShapingPbID].boSelect THEN
	                #internal.panel[#PB_Configuration.itLeftSelPbID].boAborted := #EQintHeatL."to".boStatusAbortedEQ OR #EQintHeatL."to".boStatusAbortedShape;
	                #internal.panel[#PB_Configuration.itLeftSelPbID].boHeld := #EQintHeatL."to".boStatusHeldEQ OR #EQintHeatL."to".boStatusHeldShape;

	                #internal.panel[#PB_Configuration.itOnOffSelPbID].boOnPos := #EQintHeatL."to".boPosShape;
	                #internal.panel[#PB_Configuration.itOnOffSelPbID].boMoving := #EQintHeatL."to".boActiveShape;
	                #internal.panel[#PB_Configuration.itOnOffSelPbID].boEnable := #EQintHeatL."to".boEnaShape OR #internal.panel[#PB_Configuration.itOnOffSelPbID].boMoving OR #internal.panel[#PB_Configuration.itOnOffSelPbID].boOnPos;

	                #EQintHeatL.from.boCmdShape := #internal.panel[#PB_Configuration.itOnOffSelPbID].boCmdOn;
	            END_IF;

	            // Drainage: manual commands
	            IF #internal.panel[#PB_Configuration.itDrainPbID].boSelect THEN
	                #internal.panel[#PB_Configuration.itLeftSelPbID].boAborted := #EQintHeatL."to".boStatusAbortedDrain;
	                #internal.panel[#PB_Configuration.itLeftSelPbID].boHeld := #EQintHeatL."to".boStatusHeldDrain;

	                #internal.panel[#PB_Configuration.itOnOffSelPbID].boOnPos := #EQintHeatL."to".boPosDrain;
	                #internal.panel[#PB_Configuration.itOnOffSelPbID].boMoving := #EQintHeatL."to".boActiveDrain;
	                #internal.panel[#PB_Configuration.itOnOffSelPbID].boEnable := #EQintHeatL."to".boEnaDrain OR #internal.panel[#PB_Configuration.itOnOffSelPbID].boMoving OR #internal.panel[#PB_Configuration.itOnOffSelPbID].boOnPos;

	                #EQintHeatL.from.boCmdDrain := #internal.panel[#PB_Configuration.itOnOffSelPbID].boCmdOn;
	            END_IF;

	            // Vacuum: manual commands
	            IF #internal.panel[#PB_Configuration.itVacuumPbID].boSelect THEN
	                #internal.panel[#PB_Configuration.itLeftSelPbID].boAborted := #EQintHeatL."to".boStatusAbortedVacuum;
	                #internal.panel[#PB_Configuration.itLeftSelPbID].boHeld := #EQintHeatL."to".boStatusHeldVacuum;

	                #internal.panel[#PB_Configuration.itOnOffSelPbID].boOnPos := #EQintHeatL."to".boPosVacuum;
	                #internal.panel[#PB_Configuration.itOnOffSelPbID].boMoving := #EQintHeatL."to".boActiveVacuum;
	                #internal.panel[#PB_Configuration.itOnOffSelPbID].boEnable := #EQintHeatL."to".boEnaVacuum OR #internal.panel[#PB_Configuration.itOnOffSelPbID].boMoving OR #internal.panel[#PB_Configuration.itOnOffSelPbID].boOnPos;

	                #EQintHeatL.from.boCmdVacuum := #internal.panel[#PB_Configuration.itOnOffSelPbID].boCmdOn;
	            END_IF;

	            // Enable push-buttons
	            #internal.panel[#PB_Configuration.itExtHeatingPbID].boEnable := TRUE;

	        END_IF;

	        IF (#internal.boManSelOnHeatingR OR #internal.boSetupSelOnHeatingR OR #internal.boSetupProcActiveR) AND #internal.panel[#PB_Configuration.itRightSelPbID].boSelect THEN
	            // Enable push-buttons
	            #internal.panel[#PB_Configuration.itShapingPbID].boEnable := TRUE;
	            #internal.panel[#PB_Configuration.itDrainPbID].boEnable := TRUE;
	            #internal.panel[#PB_Configuration.itVacuumPbID].boEnable := TRUE;

	            // Modules fault & warning
	            #internal.panel[#PB_Configuration.itShapingPbID].boAborted := #EQintHeatR."to".boStatusAbortedEQ OR #EQintHeatR."to".boStatusAbortedShape;
	            #internal.panel[#PB_Configuration.itDrainPbID].boAborted := #EQintHeatR."to".boStatusAbortedDrain;
	            #internal.panel[#PB_Configuration.itVacuumPbID].boAborted := #EQintHeatR."to".boStatusAbortedVacuum;
	            #internal.panel[#PB_Configuration.itShapingPbID].boHeld := #EQintHeatR."to".boStatusHeldEQ OR #EQintHeatR."to".boStatusHeldShape;
	            #internal.panel[#PB_Configuration.itDrainPbID].boHeld := #EQintHeatR."to".boStatusHeldDrain;
	            #internal.panel[#PB_Configuration.itVacuumPbID].boHeld := #EQintHeatR."to".boStatusHeldVacuum;

	            // Shaping: manual commands
	            IF #internal.panel[#PB_Configuration.itShapingPbID].boSelect THEN
	                #internal.panel[#PB_Configuration.itRightSelPbID].boAborted := #EQintHeatR."to".boStatusAbortedEQ OR #EQintHeatR."to".boStatusAbortedShape;
	                #internal.panel[#PB_Configuration.itRightSelPbID].boHeld := #EQintHeatR."to".boStatusHeldEQ OR #EQintHeatR."to".boStatusHeldShape;

	                #internal.panel[#PB_Configuration.itOnOffSelPbID].boOnPos := #EQintHeatR."to".boPosShape;
	                #internal.panel[#PB_Configuration.itOnOffSelPbID].boMoving := #EQintHeatR."to".boActiveShape;
	                #internal.panel[#PB_Configuration.itOnOffSelPbID].boEnable := #EQintHeatR."to".boEnaShape OR #internal.panel[#PB_Configuration.itOnOffSelPbID].boMoving OR #internal.panel[#PB_Configuration.itOnOffSelPbID].boOnPos;

	                #EQintHeatR.from.boCmdShape := #internal.panel[#PB_Configuration.itOnOffSelPbID].boCmdOn;
	            END_IF;

	            // Drainage: manual commands
	            IF #internal.panel[#PB_Configuration.itDrainPbID].boSelect THEN
	                #internal.panel[#PB_Configuration.itRightSelPbID].boAborted := #EQintHeatR."to".boStatusAbortedDrain;
	                #internal.panel[#PB_Configuration.itRightSelPbID].boHeld := #EQintHeatR."to".boStatusHeldDrain;

	                #internal.panel[#PB_Configuration.itOnOffSelPbID].boOnPos := #EQintHeatR."to".boPosDrain;
	                #internal.panel[#PB_Configuration.itOnOffSelPbID].boMoving := #EQintHeatR."to".boActiveDrain;
	                #internal.panel[#PB_Configuration.itOnOffSelPbID].boEnable := #EQintHeatR."to".boEnaDrain OR #internal.panel[#PB_Configuration.itOnOffSelPbID].boMoving OR #internal.panel[#PB_Configuration.itOnOffSelPbID].boOnPos;

	                #EQintHeatR.from.boCmdDrain := #internal.panel[#PB_Configuration.itOnOffSelPbID].boCmdOn;
	            END_IF;

	            // Vacuum: manual commands
	            IF #internal.panel[#PB_Configuration.itVacuumPbID].boSelect THEN
	                #internal.panel[#PB_Configuration.itRightSelPbID].boAborted := #EQintHeatR."to".boStatusAbortedVacuum;
	                #internal.panel[#PB_Configuration.itRightSelPbID].boHeld := #EQintHeatR."to".boStatusHeldVacuum;

	                #internal.panel[#PB_Configuration.itOnOffSelPbID].boOnPos := #EQintHeatR."to".boPosVacuum;
	                #internal.panel[#PB_Configuration.itOnOffSelPbID].boMoving := #EQintHeatR."to".boActiveVacuum;
	                #internal.panel[#PB_Configuration.itOnOffSelPbID].boEnable := #EQintHeatR."to".boEnaVacuum OR #internal.panel[#PB_Configuration.itOnOffSelPbID].boMoving OR #internal.panel[#PB_Configuration.itOnOffSelPbID].boOnPos;

	                #EQintHeatR.from.boCmdVacuum := #internal.panel[#PB_Configuration.itOnOffSelPbID].boCmdOn;
	            END_IF;

	            // Enable push-buttons
	            #internal.panel[#PB_Configuration.itExtHeatingPbID].boEnable := TRUE;

	        END_IF;

	        IF ((#internal.boManSelOnHeatingL OR #internal.boSetupSelOnHeatingL OR #internal.boSetupProcActiveL) AND #internal.panel[#PB_Configuration.itLeftSelPbID].boSelect) AND
	            ((#internal.boManSelOnHeatingR OR #internal.boSetupSelOnHeatingR OR #internal.boSetupProcActiveR) AND #internal.panel[#PB_Configuration.itRightSelPbID].boSelect) THEN
	            // Enable push-buttons
	            #internal.panel[#PB_Configuration.itShapingPbID].boEnable := TRUE;
	            #internal.panel[#PB_Configuration.itDrainPbID].boEnable := TRUE;
	            #internal.panel[#PB_Configuration.itVacuumPbID].boEnable := TRUE;

	            // Modules fault & warning
	            #internal.panel[#PB_Configuration.itShapingPbID].boAborted := #EQintHeatL."to".boStatusAbortedEQ OR #EQintHeatL."to".boStatusAbortedShape OR #EQintHeatR."to".boStatusAbortedEQ OR #EQintHeatR."to".boStatusAbortedShape;
	            #internal.panel[#PB_Configuration.itDrainPbID].boAborted := #EQintHeatL."to".boStatusAbortedDrain OR #EQintHeatR."to".boStatusAbortedDrain;
	            #internal.panel[#PB_Configuration.itVacuumPbID].boAborted := #EQintHeatL."to".boStatusAbortedVacuum OR #EQintHeatR."to".boStatusAbortedVacuum;
	            #internal.panel[#PB_Configuration.itShapingPbID].boHeld := #EQintHeatL."to".boStatusHeldEQ OR #EQintHeatL."to".boStatusHeldShape OR #EQintHeatR."to".boStatusHeldEQ OR #EQintHeatR."to".boStatusHeldShape;
	            #internal.panel[#PB_Configuration.itDrainPbID].boHeld := #EQintHeatL."to".boStatusHeldDrain OR #EQintHeatR."to".boStatusHeldDrain;
	            #internal.panel[#PB_Configuration.itVacuumPbID].boHeld := #EQintHeatL."to".boStatusHeldVacuum OR #EQintHeatR."to".boStatusHeldVacuum;

	            // Shaping: manual commands
	            IF #internal.panel[#PB_Configuration.itShapingPbID].boSelect THEN
	                #internal.panel[#PB_Configuration.itOnOffSelPbID].boOnPos := #EQintHeatL."to".boPosShape AND #EQintHeatR."to".boPosShape;
	                #internal.panel[#PB_Configuration.itOnOffSelPbID].boMoving := #EQintHeatL."to".boActiveShape OR #EQintHeatR."to".boActiveShape;
	                #internal.panel[#PB_Configuration.itOnOffSelPbID].boEnable := #EQintHeatL."to".boEnaShape OR #EQintHeatR."to".boEnaShape OR #internal.panel[#PB_Configuration.itOnOffSelPbID].boMoving OR #internal.panel[#PB_Configuration.itOnOffSelPbID].boOnPos;
	            END_IF;

	            // Drainage: manual commands
	            IF #internal.panel[#PB_Configuration.itDrainPbID].boSelect THEN
	                #internal.panel[#PB_Configuration.itOnOffSelPbID].boOnPos := #EQintHeatL."to".boPosDrain AND #EQintHeatR."to".boPosDrain;
	                #internal.panel[#PB_Configuration.itOnOffSelPbID].boMoving := #EQintHeatL."to".boActiveDrain OR #EQintHeatR."to".boActiveDrain;
	                #internal.panel[#PB_Configuration.itOnOffSelPbID].boEnable := #EQintHeatL."to".boEnaDrain OR #EQintHeatR."to".boEnaDrain OR #internal.panel[#PB_Configuration.itOnOffSelPbID].boMoving OR #internal.panel[#PB_Configuration.itOnOffSelPbID].boOnPos;
	            END_IF;

	            // Vacuum: manual commands
	            IF #internal.panel[#PB_Configuration.itVacuumPbID].boSelect THEN
	                #internal.panel[#PB_Configuration.itOnOffSelPbID].boOnPos := #EQintHeatL."to".boPosVacuum AND #EQintHeatR."to".boPosVacuum;
	                #internal.panel[#PB_Configuration.itOnOffSelPbID].boMoving := #EQintHeatL."to".boActiveVacuum OR #EQintHeatR."to".boActiveVacuum;
	                #internal.panel[#PB_Configuration.itOnOffSelPbID].boEnable := #EQintHeatL."to".boEnaVacuum OR #EQintHeatR."to".boEnaVacuum OR #internal.panel[#PB_Configuration.itOnOffSelPbID].boMoving OR #internal.panel[#PB_Configuration.itOnOffSelPbID].boOnPos;
	            END_IF;

	            // Enable push-buttons
	            #internal.panel[#PB_Configuration.itExtHeatingPbID].boEnable := TRUE;

